REGION Network 2: ADD A STEP
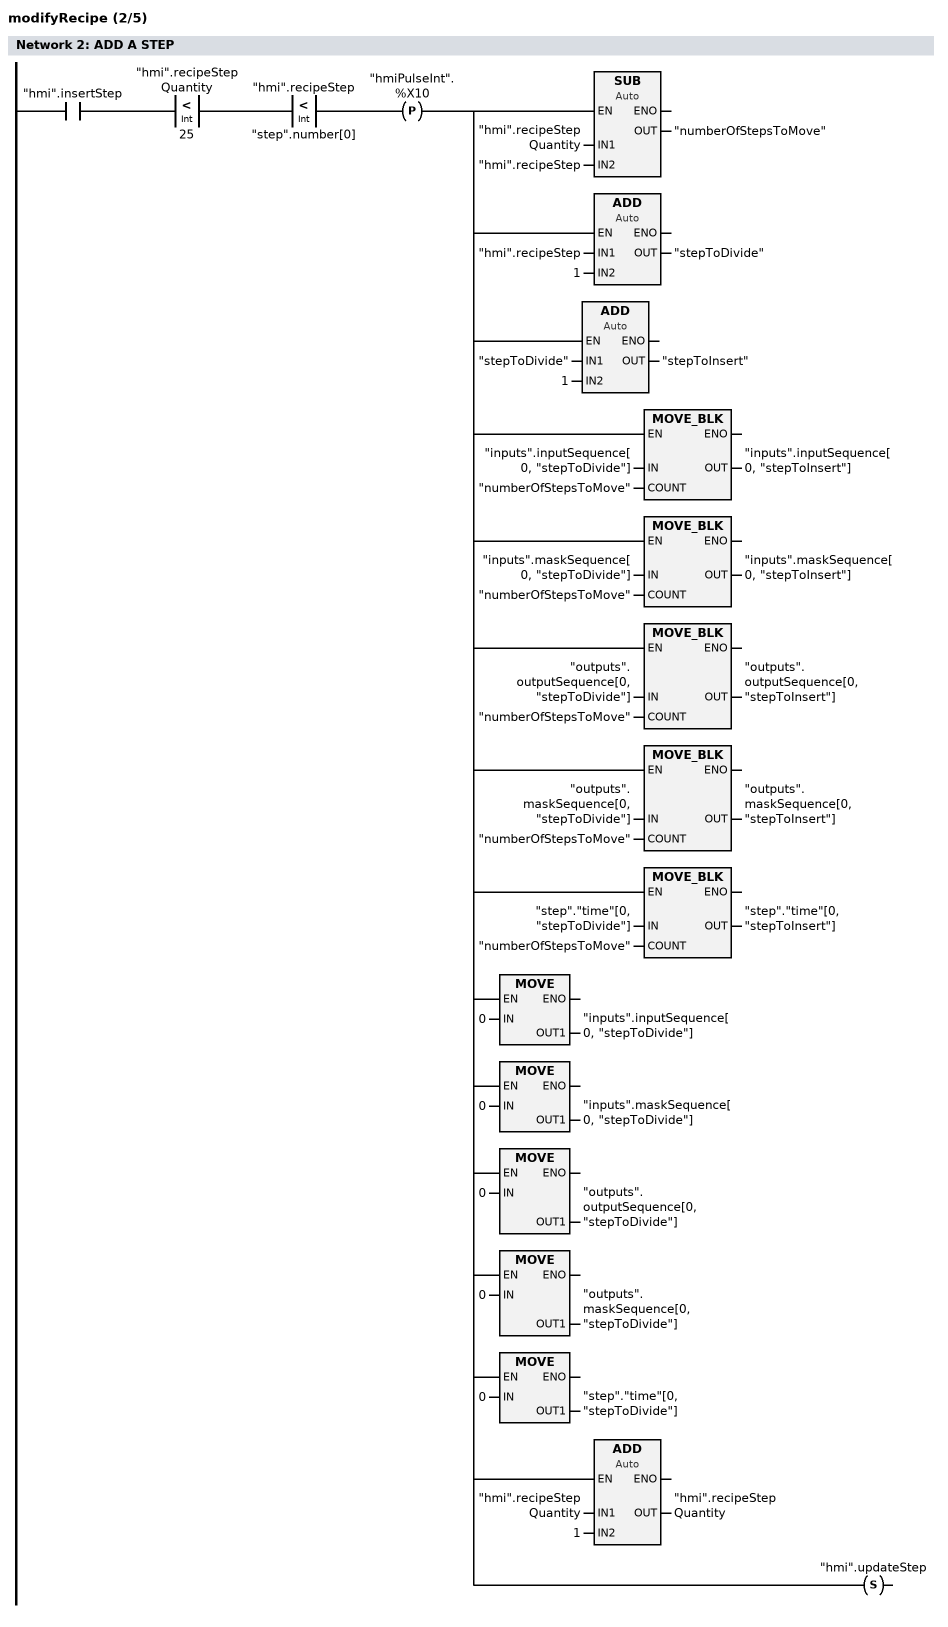
   #_w1 := "hmi".insertStep AND ("hmi".recipeStepQuantity < 25) AND ("hmi".recipeStep < "step".number[0]);
   #_w2 := #_w1 AND NOT "hmiPulseInt".%X10;   // rising edge
   "hmiPulseInt".%X10 := #_w1;
   IF #_w2 THEN
       "numberOfStepsToMove" := "hmi".recipeStepQuantity - "hmi".recipeStep;
       "stepToDivide" := "hmi".recipeStep + 1;
       "stepToInsert" := "stepToDivide" + 1;
       MOVE_BLK(IN := "inputs".inputSequence[0, "stepToDivide"],
                COUNT := "numberOfStepsToMove",
                OUT => "inputs".inputSequence[0, "stepToInsert"]);
       MOVE_BLK(IN := "inputs".maskSequence[0, "stepToDivide"],
                COUNT := "numberOfStepsToMove",
                OUT => "inputs".maskSequence[0, "stepToInsert"]);
       MOVE_BLK(IN := "outputs".outputSequence[0, "stepToDivide"],
                COUNT := "numberOfStepsToMove",
                OUT => "outputs".outputSequence[0, "stepToInsert"]);
       MOVE_BLK(IN := "outputs".maskSequence[0, "stepToDivide"],
                COUNT := "numberOfStepsToMove",
                OUT => "outputs".maskSequence[0, "stepToInsert"]);
       MOVE_BLK(IN := "step"."time"[0, "stepToDivide"],
                COUNT := "numberOfStepsToMove",
                OUT => "step"."time"[0, "stepToInsert"]);
       "inputs".inputSequence[0, "stepToDivide"] := 0;
       "inputs".maskSequence[0, "stepToDivide"] := 0;
       "outputs".outputSequence[0, "stepToDivide"] := 0;
       "outputs".maskSequence[0, "stepToDivide"] := 0;
       "step"."time"[0, "stepToDivide"] := 0;
       "hmi".recipeStepQuantity := "hmi".recipeStepQuantity + 1;
       "hmi".updateStep := TRUE;
   END_IF;
END_REGION

REGION Network 3: COPY A STEP
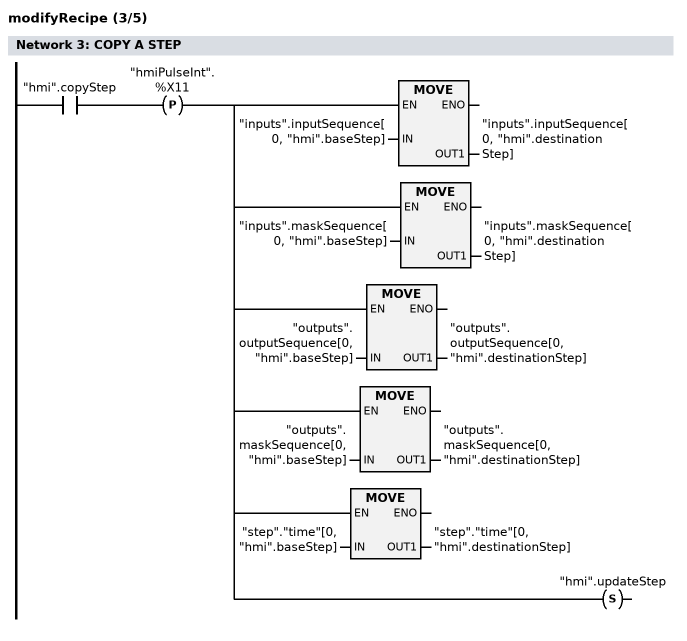
   RUNG wire#powerrail
      Contact( "hmi".copyStep )
      P_Trig( "hmiPulseInt".%X11 )
      wire#w1
      Move(in := "inputs".inputSequence[0, "hmi".baseStep], out1 => "inputs".inputSequence[0, "hmi".destinationStep])
   END_RUNG
   RUNG wire#w1
      Move(in := "inputs".maskSequence[0, "hmi".baseStep], out1 => "inputs".maskSequence[0, "hmi".destinationStep])
   END_RUNG
   RUNG wire#w1
      Move(in := "outputs".outputSequence[0, "hmi".baseStep], out1 => "outputs".outputSequence[0, "hmi".destinationStep])
   END_RUNG
   RUNG wire#w1
      Move(in := "outputs".maskSequence[0, "hmi".baseStep], out1 => "outputs".maskSequence[0, "hmi".destinationStep])
   END_RUNG
   RUNG wire#w1
      Move(in := "step"."time"[0, "hmi".baseStep], out1 => "step"."time"[0, "hmi".destinationStep])
   END_RUNG
   RUNG wire#w1
      S_Coil( "hmi".updateStep )
   END_RUNG
   // the same network as SCL:
   #_w1 := "hmi".copyStep AND NOT "hmiPulseInt".%X11;   // rising edge
   "hmiPulseInt".%X11 := "hmi".copyStep;
   IF #_w1 THEN
       "inputs".inputSequence[0, "hmi".destinationStep] := "inputs".inputSequence[0, "hmi".baseStep];
       "inputs".maskSequence[0, "hmi".destinationStep] := "inputs".maskSequence[0, "hmi".baseStep];
       "outputs".outputSequence[0, "hmi".destinationStep] := "outputs".outputSequence[0, "hmi".baseStep];
       "outputs".maskSequence[0, "hmi".destinationStep] := "outputs".maskSequence[0, "hmi".baseStep];
       "step"."time"[0, "hmi".destinationStep] := "step"."time"[0, "hmi".baseStep];
       "hmi".updateStep := TRUE;
   END_IF;
END_REGION

REGION Network 4: COPY SEQUENCE (COPY PART NUMBER)
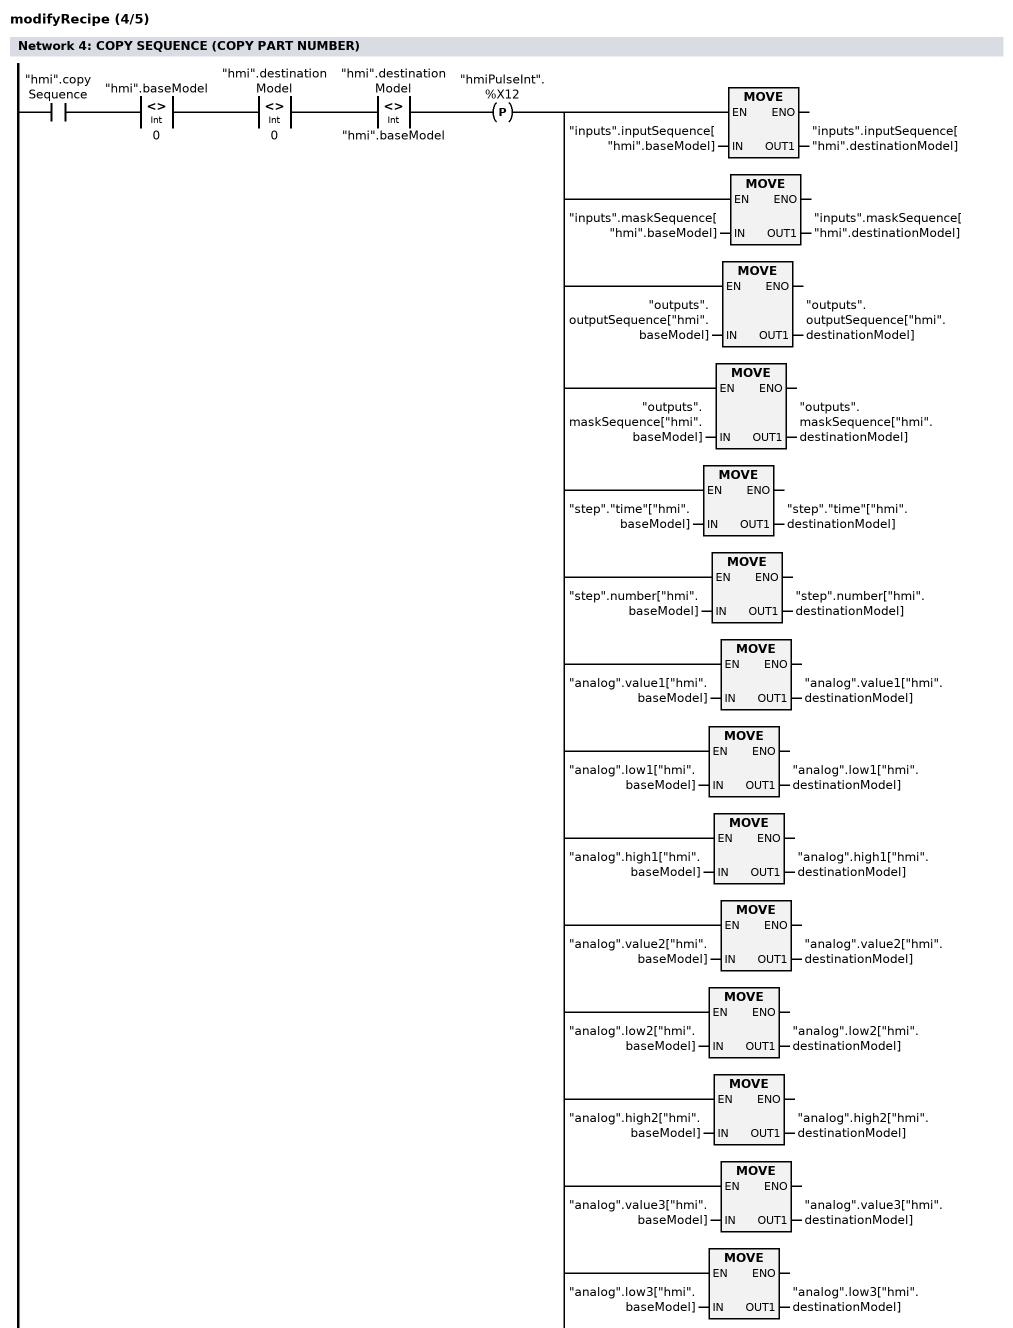
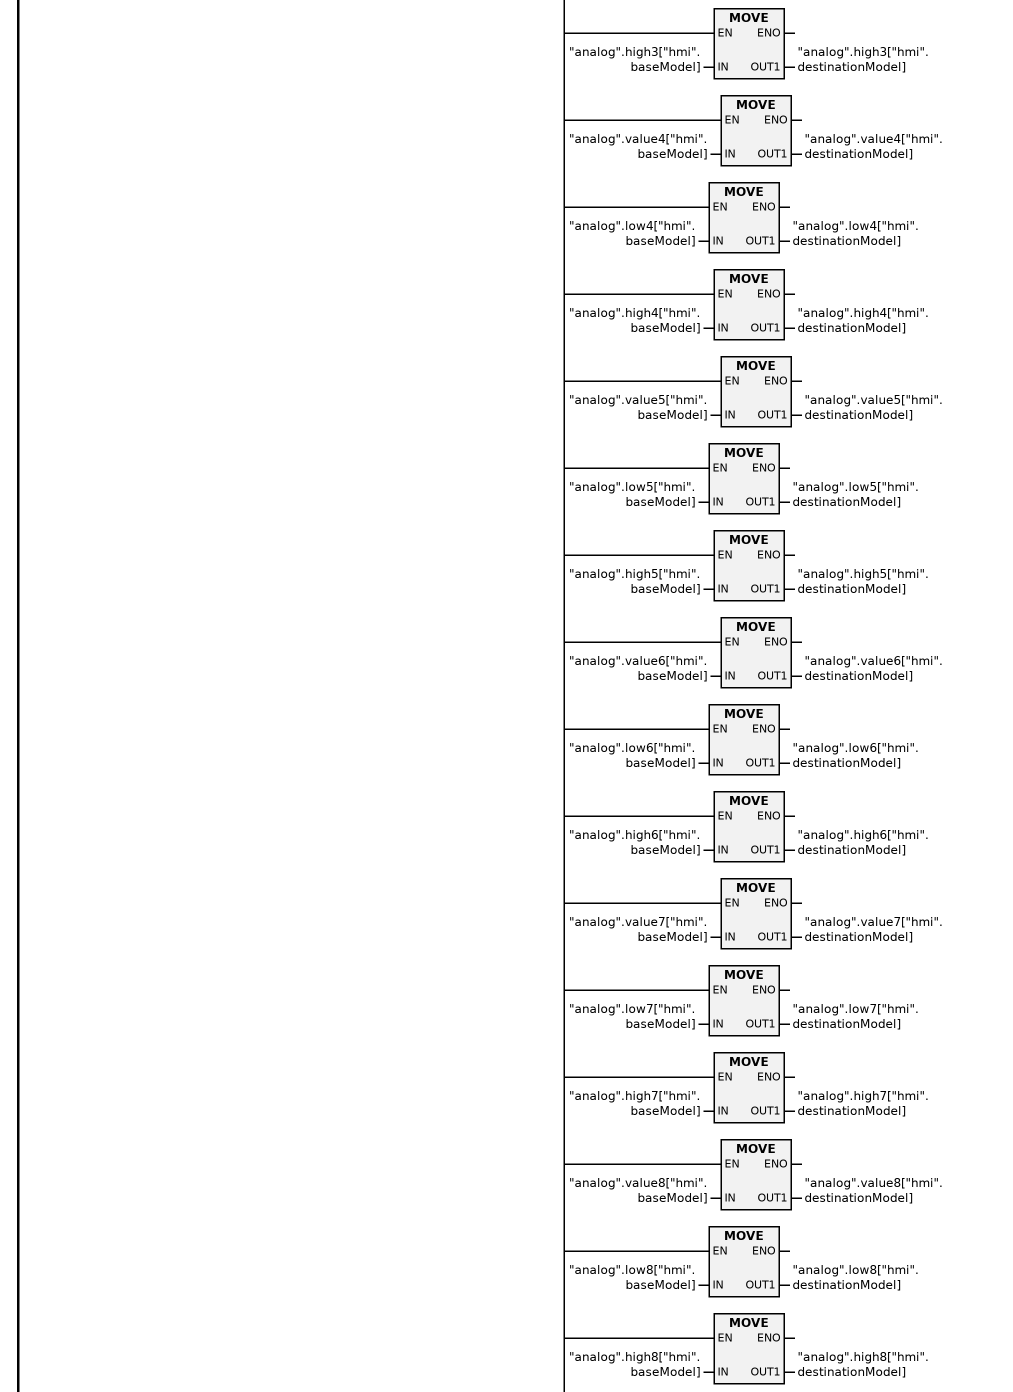
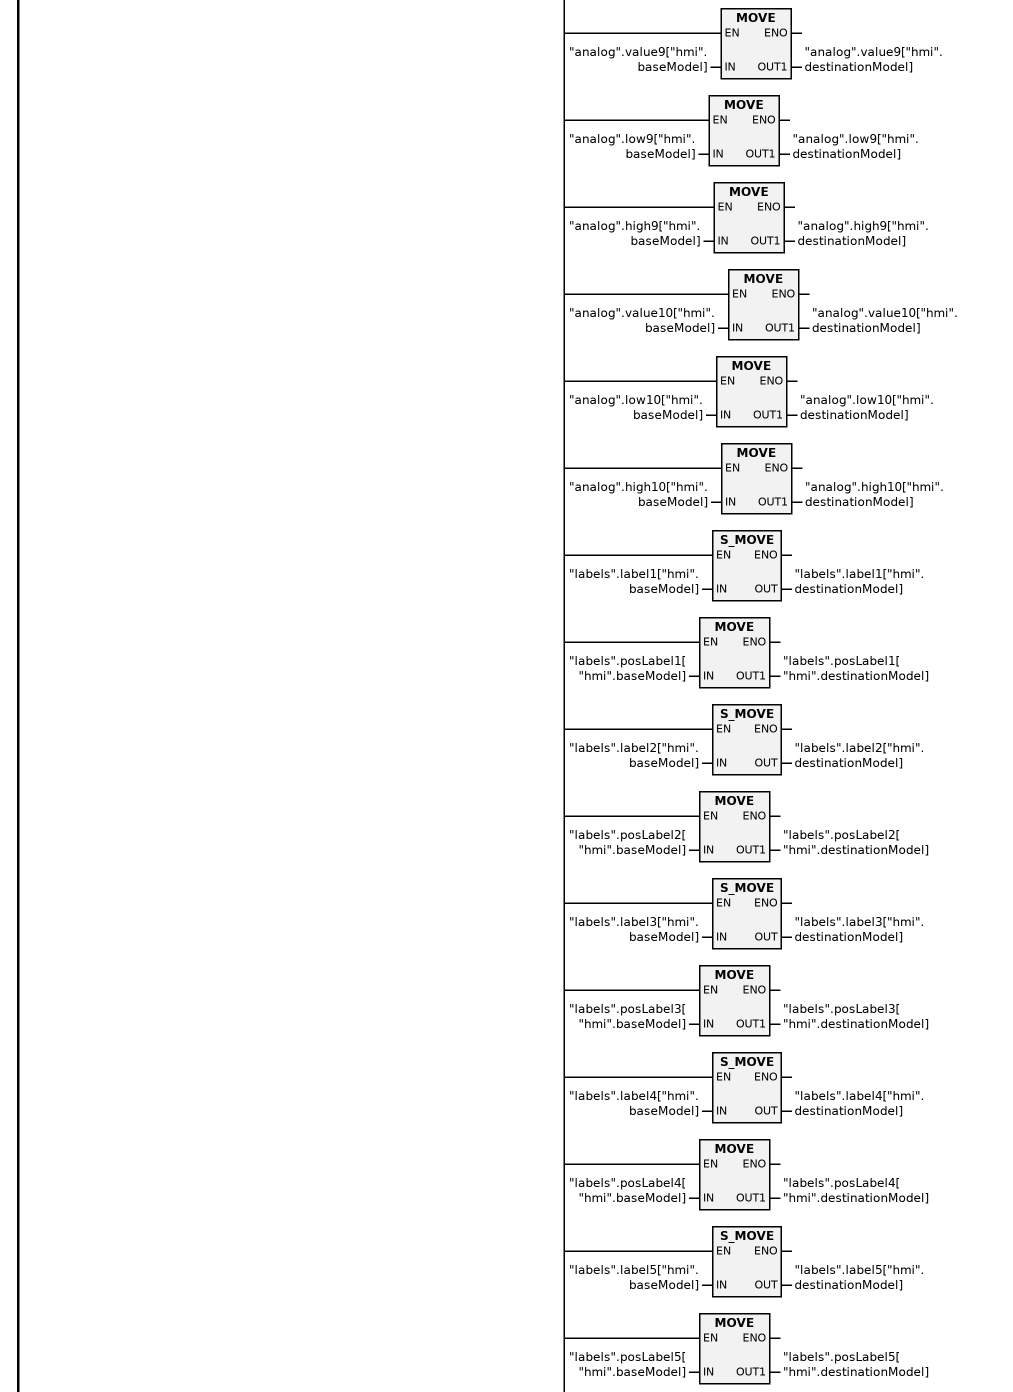
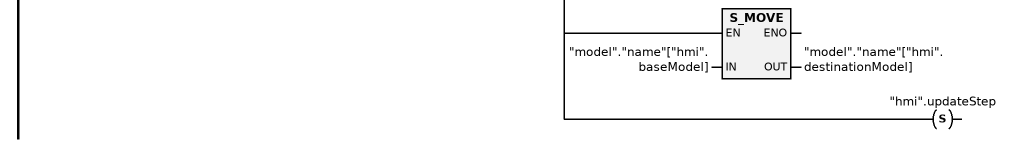
   RUNG wire#powerrail
      Contact( "hmi".copySequence )
      { S7_Templates := "SrcType := Int" } NE_Contact(in1 := "hmi".baseModel, in2 := 0)
      { S7_Templates := "SrcType := Int" } NE_Contact(in1 := "hmi".destinationModel, in2 := 0)
      { S7_Templates := "SrcType := Int" } NE_Contact(in1 := "hmi".destinationModel, in2 := "hmi".baseModel)
      P_Trig( "hmiPulseInt".%X12 )
      wire#w1
      Move(in := "inputs".inputSequence["hmi".baseModel], out1 => "inputs".inputSequence["hmi".destinationModel])
   END_RUNG
   RUNG wire#w1
      Move(in := "inputs".maskSequence["hmi".baseModel], out1 => "inputs".maskSequence["hmi".destinationModel])
   END_RUNG
   RUNG wire#w1
      Move(in := "outputs".outputSequence["hmi".baseModel], out1 => "outputs".outputSequence["hmi".destinationModel])
   END_RUNG
   RUNG wire#w1
      Move(in := "outputs".maskSequence["hmi".baseModel], out1 => "outputs".maskSequence["hmi".destinationModel])
   END_RUNG
   RUNG wire#w1
      Move(in := "step"."time"["hmi".baseModel], out1 => "step"."time"["hmi".destinationModel])
   END_RUNG
   RUNG wire#w1
      Move(in := "step".number["hmi".baseModel], out1 => "step".number["hmi".destinationModel])
   END_RUNG
   RUNG wire#w1
      Move(in := "analog".value1["hmi".baseModel], out1 => "analog".value1["hmi".destinationModel])
   END_RUNG
   RUNG wire#w1
      Move(in := "analog".low1["hmi".baseModel], out1 => "analog".low1["hmi".destinationModel])
   END_RUNG
   RUNG wire#w1
      Move(in := "analog".high1["hmi".baseModel], out1 => "analog".high1["hmi".destinationModel])
   END_RUNG
   RUNG wire#w1
      Move(in := "analog".value2["hmi".baseModel], out1 => "analog".value2["hmi".destinationModel])
   END_RUNG
   RUNG wire#w1
      Move(in := "analog".low2["hmi".baseModel], out1 => "analog".low2["hmi".destinationModel])
   END_RUNG
   RUNG wire#w1
      Move(in := "analog".high2["hmi".baseModel], out1 => "analog".high2["hmi".destinationModel])
   END_RUNG
   RUNG wire#w1
      Move(in := "analog".value3["hmi".baseModel], out1 => "analog".value3["hmi".destinationModel])
   END_RUNG
   RUNG wire#w1
      Move(in := "analog".low3["hmi".baseModel], out1 => "analog".low3["hmi".destinationModel])
   END_RUNG
   RUNG wire#w1
      Move(in := "analog".high3["hmi".baseModel], out1 => "analog".high3["hmi".destinationModel])
   END_RUNG
   RUNG wire#w1
      Move(in := "analog".value4["hmi".baseModel], out1 => "analog".value4["hmi".destinationModel])
   END_RUNG
   RUNG wire#w1
      Move(in := "analog".low4["hmi".baseModel], out1 => "analog".low4["hmi".destinationModel])
   END_RUNG
   RUNG wire#w1
      Move(in := "analog".high4["hmi".baseModel], out1 => "analog".high4["hmi".destinationModel])
   END_RUNG
   RUNG wire#w1
      Move(in := "analog".value5["hmi".baseModel], out1 => "analog".value5["hmi".destinationModel])
   END_RUNG
   RUNG wire#w1
      Move(in := "analog".low5["hmi".baseModel], out1 => "analog".low5["hmi".destinationModel])
   END_RUNG
   RUNG wire#w1
      Move(in := "analog".high5["hmi".baseModel], out1 => "analog".high5["hmi".destinationModel])
   END_RUNG
   RUNG wire#w1
      Move(in := "analog".value6["hmi".baseModel], out1 => "analog".value6["hmi".destinationModel])
   END_RUNG
   RUNG wire#w1
      Move(in := "analog".low6["hmi".baseModel], out1 => "analog".low6["hmi".destinationModel])
   END_RUNG
   RUNG wire#w1
      Move(in := "analog".high6["hmi".baseModel], out1 => "analog".high6["hmi".destinationModel])
   END_RUNG
   RUNG wire#w1
      Move(in := "analog".value7["hmi".baseModel], out1 => "analog".value7["hmi".destinationModel])
   END_RUNG
   RUNG wire#w1
      Move(in := "analog".low7["hmi".baseModel], out1 => "analog".low7["hmi".destinationModel])
   END_RUNG
   RUNG wire#w1
      Move(in := "analog".high7["hmi".baseModel], out1 => "analog".high7["hmi".destinationModel])
   END_RUNG
   RUNG wire#w1
      Move(in := "analog".value8["hmi".baseModel], out1 => "analog".value8["hmi".destinationModel])
   END_RUNG
   RUNG wire#w1
      Move(in := "analog".low8["hmi".baseModel], out1 => "analog".low8["hmi".destinationModel])
   END_RUNG
   RUNG wire#w1
      Move(in := "analog".high8["hmi".baseModel], out1 => "analog".high8["hmi".destinationModel])
   END_RUNG
   RUNG wire#w1
      Move(in := "analog".value9["hmi".baseModel], out1 => "analog".value9["hmi".destinationModel])
   END_RUNG
   RUNG wire#w1
      Move(in := "analog".low9["hmi".baseModel], out1 => "analog".low9["hmi".destinationModel])
   END_RUNG
   RUNG wire#w1
      Move(in := "analog".high9["hmi".baseModel], out1 => "analog".high9["hmi".destinationModel])
   END_RUNG
   RUNG wire#w1
      Move(in := "analog".value10["hmi".baseModel], out1 => "analog".value10["hmi".destinationModel])
   END_RUNG
   RUNG wire#w1
      Move(in := "analog".low10["hmi".baseModel], out1 => "analog".low10["hmi".destinationModel])
   END_RUNG
   RUNG wire#w1
      Move(in := "analog".high10["hmi".baseModel], out1 => "analog".high10["hmi".destinationModel])
   END_RUNG
   RUNG wire#w1
      S_Move(in := "labels".label1["hmi".baseModel], out => "labels".label1["hmi".destinationModel])
   END_RUNG
   RUNG wire#w1
      Move(in := "labels".posLabel1["hmi".baseModel], out1 => "labels".posLabel1["hmi".destinationModel])
   END_RUNG
   RUNG wire#w1
      S_Move(in := "labels".label2["hmi".baseModel], out => "labels".label2["hmi".destinationModel])
   END_RUNG
   RUNG wire#w1
      Move(in := "labels".posLabel2["hmi".baseModel], out1 => "labels".posLabel2["hmi".destinationModel])
   END_RUNG
   RUNG wire#w1
      S_Move(in := "labels".label3["hmi".baseModel], out => "labels".label3["hmi".destinationModel])
   END_RUNG
   RUNG wire#w1
      Move(in := "labels".posLabel3["hmi".baseModel], out1 => "labels".posLabel3["hmi".destinationModel])
   END_RUNG
   RUNG wire#w1
      S_Move(in := "labels".label4["hmi".baseModel], out => "labels".label4["hmi".destinationModel])
   END_RUNG
   RUNG wire#w1
      Move(in := "labels".posLabel4["hmi".baseModel], out1 => "labels".posLabel4["hmi".destinationModel])
   END_RUNG
   RUNG wire#w1
      S_Move(in := "labels".label5["hmi".baseModel], out => "labels".label5["hmi".destinationModel])
   END_RUNG
   RUNG wire#w1
      Move(in := "labels".posLabel5["hmi".baseModel], out1 => "labels".posLabel5["hmi".destinationModel])
   END_RUNG
   RUNG wire#w1
      S_Move(in := "model"."name"["hmi".baseModel], out => "model"."name"["hmi".destinationModel])
   END_RUNG
   RUNG wire#w1
      S_Coil( "hmi".updateStep )
   END_RUNG
   // the same network as SCL:
   #_w1 := "hmi".copySequence AND ("hmi".baseModel <> 0) AND ("hmi".destinationModel <> 0) AND ("hmi".destinationModel <> "hmi".baseModel);
   #_w2 := #_w1 AND NOT "hmiPulseInt".%X12;   // rising edge
   "hmiPulseInt".%X12 := #_w1;
   IF #_w2 THEN
       "inputs".inputSequence["hmi".destinationModel] := "inputs".inputSequence["hmi".baseModel];
       "inputs".maskSequence["hmi".destinationModel] := "inputs".maskSequence["hmi".baseModel];
       "outputs".outputSequence["hmi".destinationModel] := "outputs".outputSequence["hmi".baseModel];
       "outputs".maskSequence["hmi".destinationModel] := "outputs".maskSequence["hmi".baseModel];
       "step"."time"["hmi".destinationModel] := "step"."time"["hmi".baseModel];
       "step".number["hmi".destinationModel] := "step".number["hmi".baseModel];
       "analog".value1["hmi".destinationModel] := "analog".value1["hmi".baseModel];
       "analog".low1["hmi".destinationModel] := "analog".low1["hmi".baseModel];
       "analog".high1["hmi".destinationModel] := "analog".high1["hmi".baseModel];
       "analog".value2["hmi".destinationModel] := "analog".value2["hmi".baseModel];
       "analog".low2["hmi".destinationModel] := "analog".low2["hmi".baseModel];
       "analog".high2["hmi".destinationModel] := "analog".high2["hmi".baseModel];
       "analog".value3["hmi".destinationModel] := "analog".value3["hmi".baseModel];
       "analog".low3["hmi".destinationModel] := "analog".low3["hmi".baseModel];
       "analog".high3["hmi".destinationModel] := "analog".high3["hmi".baseModel];
       "analog".value4["hmi".destinationModel] := "analog".value4["hmi".baseModel];
       "analog".low4["hmi".destinationModel] := "analog".low4["hmi".baseModel];
       "analog".high4["hmi".destinationModel] := "analog".high4["hmi".baseModel];
       "analog".value5["hmi".destinationModel] := "analog".value5["hmi".baseModel];
       "analog".low5["hmi".destinationModel] := "analog".low5["hmi".baseModel];
       "analog".high5["hmi".destinationModel] := "analog".high5["hmi".baseModel];
       "analog".value6["hmi".destinationModel] := "analog".value6["hmi".baseModel];
       "analog".low6["hmi".destinationModel] := "analog".low6["hmi".baseModel];
       "analog".high6["hmi".destinationModel] := "analog".high6["hmi".baseModel];
       "analog".value7["hmi".destinationModel] := "analog".value7["hmi".baseModel];
       "analog".low7["hmi".destinationModel] := "analog".low7["hmi".baseModel];
       "analog".high7["hmi".destinationModel] := "analog".high7["hmi".baseModel];
       "analog".value8["hmi".destinationModel] := "analog".value8["hmi".baseModel];
       "analog".low8["hmi".destinationModel] := "analog".low8["hmi".baseModel];
       "analog".high8["hmi".destinationModel] := "analog".high8["hmi".baseModel];
       "analog".value9["hmi".destinationModel] := "analog".value9["hmi".baseModel];
       "analog".low9["hmi".destinationModel] := "analog".low9["hmi".baseModel];
       "analog".high9["hmi".destinationModel] := "analog".high9["hmi".baseModel];
       "analog".value10["hmi".destinationModel] := "analog".value10["hmi".baseModel];
       "analog".low10["hmi".destinationModel] := "analog".low10["hmi".baseModel];
       "analog".high10["hmi".destinationModel] := "analog".high10["hmi".baseModel];
       "labels".label1["hmi".destinationModel] := "labels".label1["hmi".baseModel];
       "labels".posLabel1["hmi".destinationModel] := "labels".posLabel1["hmi".baseModel];
       "labels".label2["hmi".destinationModel] := "labels".label2["hmi".baseModel];
       "labels".posLabel2["hmi".destinationModel] := "labels".posLabel2["hmi".baseModel];
       "labels".label3["hmi".destinationModel] := "labels".label3["hmi".baseModel];
       "labels".posLabel3["hmi".destinationModel] := "labels".posLabel3["hmi".baseModel];
       "labels".label4["hmi".destinationModel] := "labels".label4["hmi".baseModel];
       "labels".posLabel4["hmi".destinationModel] := "labels".posLabel4["hmi".baseModel];
       "labels".label5["hmi".destinationModel] := "labels".label5["hmi".baseModel];
       "labels".posLabel5["hmi".destinationModel] := "labels".posLabel5["hmi".baseModel];
       "model"."name"["hmi".destinationModel] := "model"."name"["hmi".baseModel];
       "hmi".updateStep := TRUE;
   END_IF;
END_REGION

REGION Network 5: COPY A STEP (#) FROM A PROGRAM (#) IN ANOTHER STEP (#) FROM ANOTHER PROGRAM (#)
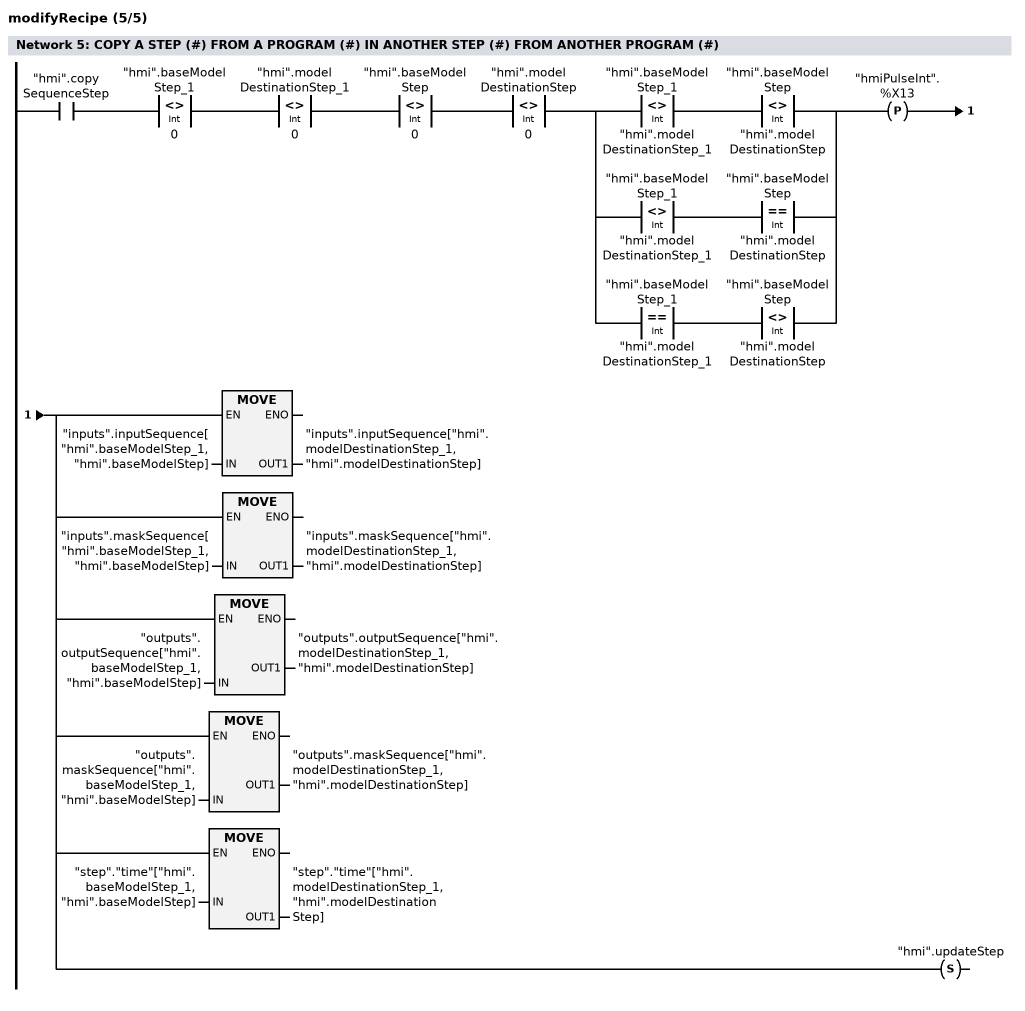
   RUNG wire#powerrail
      Contact( "hmi".copySequenceStep )
      { S7_Templates := "SrcType := Int" } NE_Contact(in1 := "hmi".baseModelStep_1, in2 := 0)
      { S7_Templates := "SrcType := Int" } NE_Contact(in1 := "hmi".modelDestinationStep_1, in2 := 0)
      { S7_Templates := "SrcType := Int" } NE_Contact(in1 := "hmi".baseModelStep, in2 := 0)
      { S7_Templates := "SrcType := Int" } NE_Contact(in1 := "hmi".modelDestinationStep, in2 := 0)
      wire#w1
      { S7_Templates := "SrcType := Int" } NE_Contact(in1 := "hmi".baseModelStep_1, in2 := "hmi".modelDestinationStep_1)
      { S7_Templates := "SrcType := Int" } NE_Contact(in1 := "hmi".baseModelStep, in2 := "hmi".modelDestinationStep)
      wire#w2
      P_Trig( "hmiPulseInt".%X13 )
      wire#w3
      Move(in := "inputs".inputSequence["hmi".baseModelStep_1, "hmi".baseModelStep], out1 => "inputs".inputSequence["hmi".modelDestinationStep_1, "hmi".modelDestinationStep])
   END_RUNG
   RUNG wire#w1
      { S7_Templates := "SrcType := Int" } NE_Contact(in1 := "hmi".baseModelStep_1, in2 := "hmi".modelDestinationStep_1)
      { S7_Templates := "SrcType := Int" } EQ_Contact(in1 := "hmi".baseModelStep, in2 := "hmi".modelDestinationStep)
   END_RUNG wire#w2
   RUNG wire#w1
      { S7_Templates := "SrcType := Int" } EQ_Contact(in1 := "hmi".baseModelStep_1, in2 := "hmi".modelDestinationStep_1)
      { S7_Templates := "SrcType := Int" } NE_Contact(in1 := "hmi".baseModelStep, in2 := "hmi".modelDestinationStep)
   END_RUNG wire#w2
   RUNG wire#w3
      Move(in := "inputs".maskSequence["hmi".baseModelStep_1, "hmi".baseModelStep], out1 => "inputs".maskSequence["hmi".modelDestinationStep_1, "hmi".modelDestinationStep])
   END_RUNG
   RUNG wire#w3
      Move(in := "outputs".outputSequence["hmi".baseModelStep_1, "hmi".baseModelStep], out1 => "outputs".outputSequence["hmi".modelDestinationStep_1, "hmi".modelDestinationStep])
   END_RUNG
   RUNG wire#w3
      Move(in := "outputs".maskSequence["hmi".baseModelStep_1, "hmi".baseModelStep], out1 => "outputs".maskSequence["hmi".modelDestinationStep_1, "hmi".modelDestinationStep])
   END_RUNG
   RUNG wire#w3
      Move(in := "step"."time"["hmi".baseModelStep_1, "hmi".baseModelStep], out1 => "step"."time"["hmi".modelDestinationStep_1, "hmi".modelDestinationStep])
   END_RUNG
   RUNG wire#w3
      S_Coil( "hmi".updateStep )
   END_RUNG
   // the same network as SCL:
   #_w1 := "hmi".copySequenceStep AND ("hmi".baseModelStep_1 <> 0) AND ("hmi".modelDestinationStep_1 <> 0) AND ("hmi".baseModelStep <> 0) AND ("hmi".modelDestinationStep <> 0) AND ((("hmi".baseModelStep_1 <> "hmi".modelDestinationStep_1) AND ("hmi".baseModelStep <> "hmi".modelDestinationStep)) OR (("hmi".baseModelStep_1 <> "hmi".modelDestinationStep_1) AND ("hmi".baseModelStep = "hmi".modelDestinationStep)) OR (("hmi".baseModelStep_1 = "hmi".modelDestinationStep_1) AND ("hmi".baseModelStep <> "hmi".modelDestinationStep)));
   #_w2 := #_w1 AND NOT "hmiPulseInt".%X13;   // rising edge
   "hmiPulseInt".%X13 := #_w1;
   IF #_w2 THEN
       "inputs".inputSequence["hmi".modelDestinationStep_1, "hmi".modelDestinationStep] := "inputs".inputSequence["hmi".baseModelStep_1, "hmi".baseModelStep];
       "inputs".maskSequence["hmi".modelDestinationStep_1, "hmi".modelDestinationStep] := "inputs".maskSequence["hmi".baseModelStep_1, "hmi".baseModelStep];
       "outputs".outputSequence["hmi".modelDestinationStep_1, "hmi".modelDestinationStep] := "outputs".outputSequence["hmi".baseModelStep_1, "hmi".baseModelStep];
       "outputs".maskSequence["hmi".modelDestinationStep_1, "hmi".modelDestinationStep] := "outputs".maskSequence["hmi".baseModelStep_1, "hmi".baseModelStep];
       "step"."time"["hmi".modelDestinationStep_1, "hmi".modelDestinationStep] := "step"."time"["hmi".baseModelStep_1, "hmi".baseModelStep];
       "hmi".updateStep := TRUE;
   END_IF;
END_REGION
END_FUNCTION

FUNCTION "inputsMapping" : Void   // FC1, LAD
{ S7_Optimized_Access := 'TRUE' }
VERSION : 0.1
// stored: AutoNumber true, IsIECCheckEnabled false, SetENOAutomatically false, UDAEnableTagReadback false
BEGIN

REGION Network 1: A00.- Clear Data
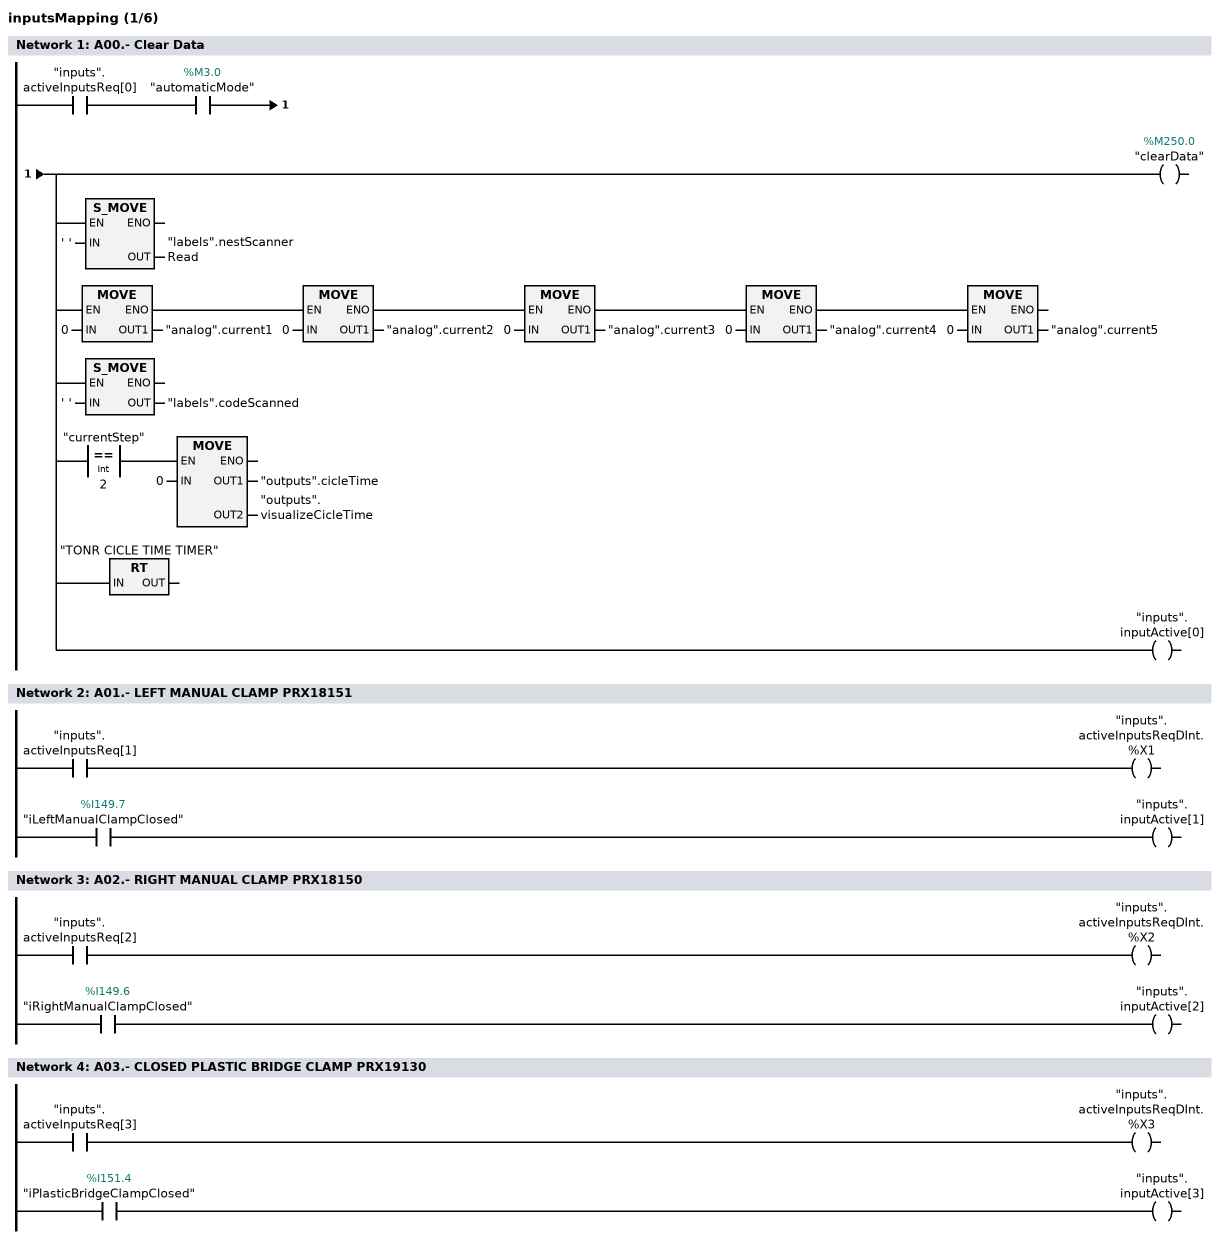
   RUNG wire#powerrail
      Contact( "inputs".activeInputsReq[0] )
      Contact( "automaticMode" )
      wire#w1
      Coil( "clearData" )
   END_RUNG
   RUNG wire#w1
      S_Move(in := ' ', out => "labels".nestScannerRead)
   END_RUNG
   RUNG wire#w1
      Move(in := 0, out1 => "analog".current1)
      Move(in := 0, out1 => "analog".current2)
      Move(in := 0, out1 => "analog".current3)
      Move(in := 0, out1 => "analog".current4)
      Move(in := 0, out1 => "analog".current5)
   END_RUNG
   RUNG wire#w1
      S_Move(in := ' ', out => "labels".codeScanned)
   END_RUNG
   RUNG wire#w1
      { S7_Templates := "SrcType := Int" } EQ_Contact(in1 := "currentStep", in2 := 2)
      Move(in := 0, out1 => "outputs".cicleTime, out2 => "outputs".visualizeCicleTime)
   END_RUNG
   RUNG wire#w1
      RT_Coil( "TONR CICLE TIME TIMER" )
   END_RUNG
   RUNG wire#w1
      Coil( "inputs".inputActive[0] )
   END_RUNG
   // the same network as SCL:
   "clearData" := "inputs".activeInputsReq[0] AND "automaticMode";
   IF "clearData" THEN
       "labels".nestScannerRead := ' ';
       "analog".current1 := 0;
       "analog".current2 := 0;
       "analog".current3 := 0;
       "analog".current4 := 0;
       "analog".current5 := 0;
       "labels".codeScanned := ' ';
   END_IF;
   IF "clearData" AND ("currentStep" = 2) THEN
       "outputs".cicleTime := 0;
       "outputs".visualizeCicleTime := 0;
   END_IF;
   IF "clearData" THEN RESET_TIMER("TONR CICLE TIME TIMER"); END_IF;
   "inputs".inputActive[0] := "clearData";
END_REGION

REGION Network 2: A01.- LEFT MANUAL CLAMP PRX18151
   RUNG wire#powerrail
      Contact( "inputs".activeInputsReq[1] )
      Coil( "inputs".activeInputsReqDInt.%X1 )
   END_RUNG
   RUNG wire#powerrail
      Contact( "iLeftManualClampClosed" )
      Coil( "inputs".inputActive[1] )
   END_RUNG
   // the same network as SCL:
   "inputs".activeInputsReqDInt.%X1 := "inputs".activeInputsReq[1];
   "inputs".inputActive[1] := "iLeftManualClampClosed";
END_REGION

REGION Network 3: A02.- RIGHT MANUAL CLAMP PRX18150
   RUNG wire#powerrail
      Contact( "inputs".activeInputsReq[2] )
      Coil( "inputs".activeInputsReqDInt.%X2 )
   END_RUNG
   RUNG wire#powerrail
      Contact( "iRightManualClampClosed" )
      Coil( "inputs".inputActive[2] )
   END_RUNG
   // the same network as SCL:
   "inputs".activeInputsReqDInt.%X2 := "inputs".activeInputsReq[2];
   "inputs".inputActive[2] := "iRightManualClampClosed";
END_REGION

REGION Network 4: A03.- CLOSED PLASTIC BRIDGE CLAMP PRX19130
   RUNG wire#powerrail
      Contact( "inputs".activeInputsReq[3] )
      Coil( "inputs".activeInputsReqDInt.%X3 )
   END_RUNG
   RUNG wire#powerrail
      Contact( "iPlasticBridgeClampClosed" )
      Coil( "inputs".inputActive[3] )
   END_RUNG
   // the same network as SCL:
   "inputs".activeInputsReqDInt.%X3 := "inputs".activeInputsReq[3];
   "inputs".inputActive[3] := "iPlasticBridgeClampClosed";
END_REGION

REGION Network 5: A04.- PLASTIC BRIDGE PRESENT PRX19090
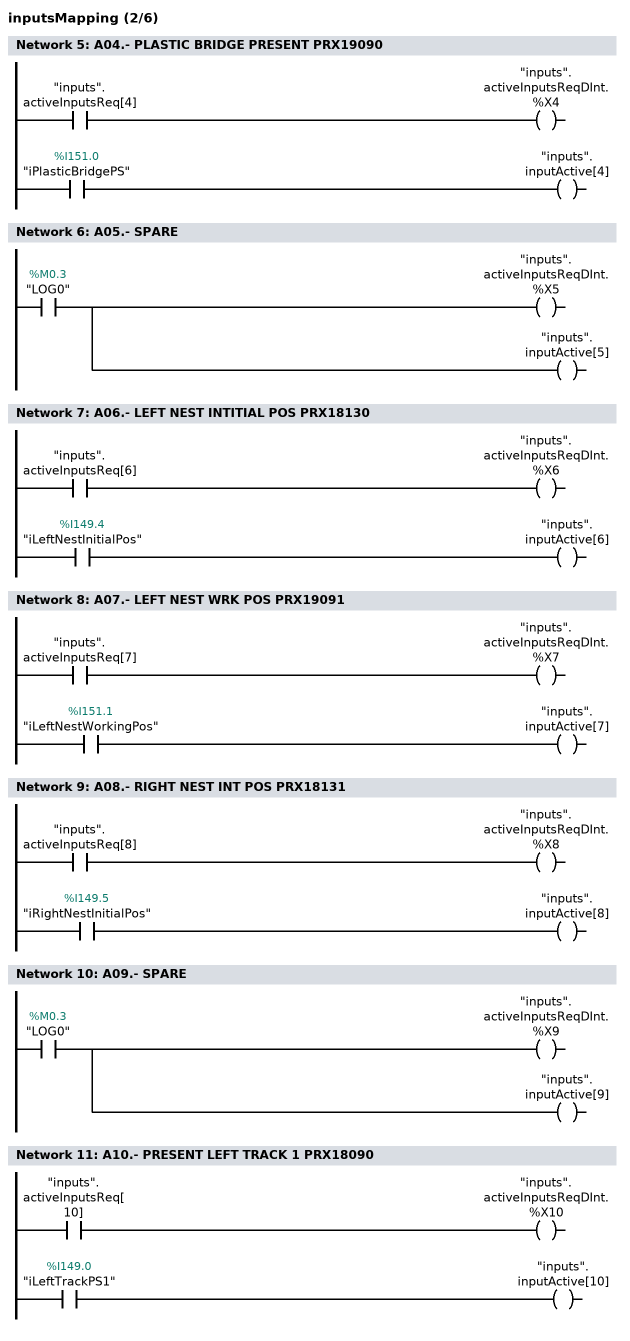
   RUNG wire#powerrail
      Contact( "inputs".activeInputsReq[4] )
      Coil( "inputs".activeInputsReqDInt.%X4 )
   END_RUNG
   RUNG wire#powerrail
      Contact( "iPlasticBridgePS" )
      Coil( "inputs".inputActive[4] )
   END_RUNG
   // the same network as SCL:
   "inputs".activeInputsReqDInt.%X4 := "inputs".activeInputsReq[4];
   "inputs".inputActive[4] := "iPlasticBridgePS";
END_REGION

REGION Network 6: A05.- SPARE
   RUNG wire#powerrail
      Contact( "LOG0" )
      wire#w1
      Coil( "inputs".activeInputsReqDInt.%X5 )
   END_RUNG
   RUNG wire#w1
      Coil( "inputs".inputActive[5] )
   END_RUNG
   // the same network as SCL:
   "inputs".activeInputsReqDInt.%X5 := "LOG0";
   "inputs".inputActive[5] := "LOG0";
END_REGION

REGION Network 7: A06.- LEFT NEST INTITIAL POS PRX18130
   RUNG wire#powerrail
      Contact( "inputs".activeInputsReq[6] )
      Coil( "inputs".activeInputsReqDInt.%X6 )
   END_RUNG
   RUNG wire#powerrail
      Contact( "iLeftNestInitialPos" )
      Coil( "inputs".inputActive[6] )
   END_RUNG
   // the same network as SCL:
   "inputs".activeInputsReqDInt.%X6 := "inputs".activeInputsReq[6];
   "inputs".inputActive[6] := "iLeftNestInitialPos";
END_REGION

REGION Network 8: A07.- LEFT NEST WRK POS PRX19091
   RUNG wire#powerrail
      Contact( "inputs".activeInputsReq[7] )
      Coil( "inputs".activeInputsReqDInt.%X7 )
   END_RUNG
   RUNG wire#powerrail
      Contact( "iLeftNestWorkingPos" )
      Coil( "inputs".inputActive[7] )
   END_RUNG
   // the same network as SCL:
   "inputs".activeInputsReqDInt.%X7 := "inputs".activeInputsReq[7];
   "inputs".inputActive[7] := "iLeftNestWorkingPos";
END_REGION

REGION Network 9: A08.- RIGHT NEST INT POS PRX18131
   RUNG wire#powerrail
      Contact( "inputs".activeInputsReq[8] )
      Coil( "inputs".activeInputsReqDInt.%X8 )
   END_RUNG
   RUNG wire#powerrail
      Contact( "iRightNestInitialPos" )
      Coil( "inputs".inputActive[8] )
   END_RUNG
   // the same network as SCL:
   "inputs".activeInputsReqDInt.%X8 := "inputs".activeInputsReq[8];
   "inputs".inputActive[8] := "iRightNestInitialPos";
END_REGION

REGION Network 10: A09.- SPARE
   RUNG wire#powerrail
      Contact( "LOG0" )
      wire#w1
      Coil( "inputs".activeInputsReqDInt.%X9 )
   END_RUNG
   RUNG wire#w1
      Coil( "inputs".inputActive[9] )
   END_RUNG
   // the same network as SCL:
   "inputs".activeInputsReqDInt.%X9 := "LOG0";
   "inputs".inputActive[9] := "LOG0";
END_REGION

REGION Network 11: A10.- PRESENT LEFT TRACK 1 PRX18090
   RUNG wire#powerrail
      Contact( "inputs".activeInputsReq[10] )
      Coil( "inputs".activeInputsReqDInt.%X10 )
   END_RUNG
   RUNG wire#powerrail
      Contact( "iLeftTrackPS1" )
      Coil( "inputs".inputActive[10] )
   END_RUNG
   // the same network as SCL:
   "inputs".activeInputsReqDInt.%X10 := "inputs".activeInputsReq[10];
   "inputs".inputActive[10] := "iLeftTrackPS1";
END_REGION

REGION Network 12: A11.- PRESENT RIGHT TRACK 1 PRX18110
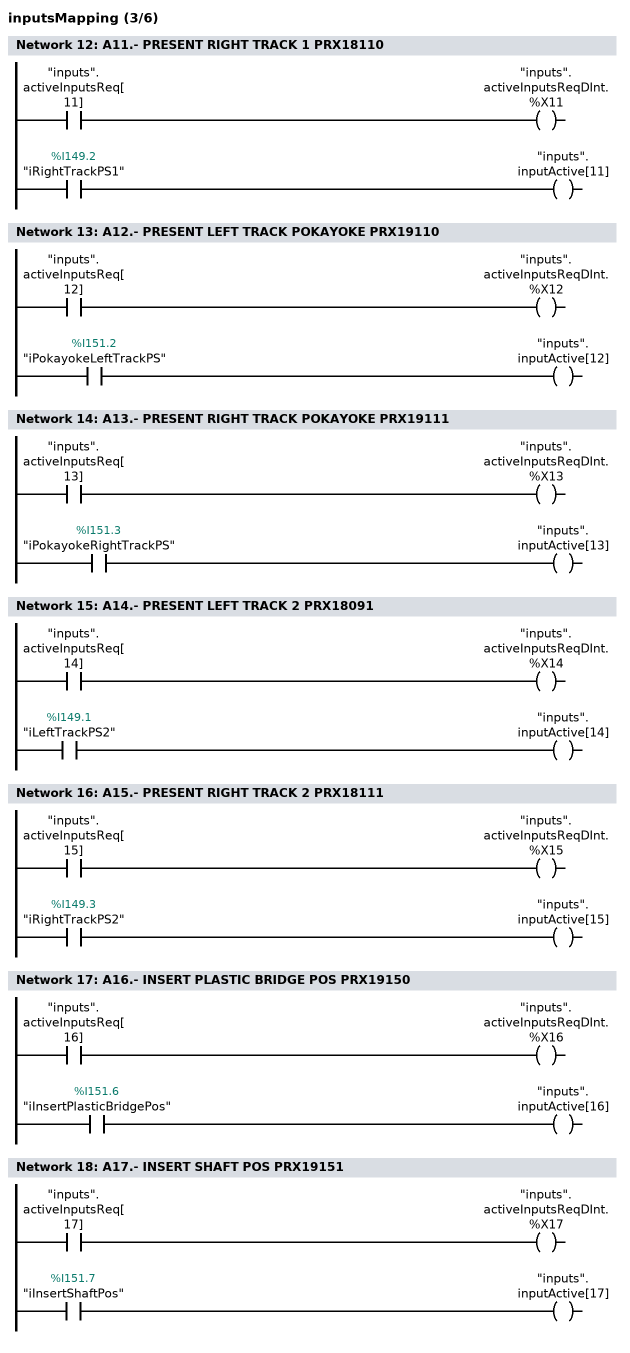
   RUNG wire#powerrail
      Contact( "inputs".activeInputsReq[11] )
      Coil( "inputs".activeInputsReqDInt.%X11 )
   END_RUNG
   RUNG wire#powerrail
      Contact( "iRightTrackPS1" )
      Coil( "inputs".inputActive[11] )
   END_RUNG
   // the same network as SCL:
   "inputs".activeInputsReqDInt.%X11 := "inputs".activeInputsReq[11];
   "inputs".inputActive[11] := "iRightTrackPS1";
END_REGION

REGION Network 13: A12.- PRESENT LEFT TRACK POKAYOKE PRX19110
   RUNG wire#powerrail
      Contact( "inputs".activeInputsReq[12] )
      Coil( "inputs".activeInputsReqDInt.%X12 )
   END_RUNG
   RUNG wire#powerrail
      Contact( "iPokayokeLeftTrackPS" )
      Coil( "inputs".inputActive[12] )
   END_RUNG
   // the same network as SCL:
   "inputs".activeInputsReqDInt.%X12 := "inputs".activeInputsReq[12];
   "inputs".inputActive[12] := "iPokayokeLeftTrackPS";
END_REGION

REGION Network 14: A13.- PRESENT RIGHT TRACK POKAYOKE PRX19111
   RUNG wire#powerrail
      Contact( "inputs".activeInputsReq[13] )
      Coil( "inputs".activeInputsReqDInt.%X13 )
   END_RUNG
   RUNG wire#powerrail
      Contact( "iPokayokeRightTrackPS" )
      Coil( "inputs".inputActive[13] )
   END_RUNG
   // the same network as SCL:
   "inputs".activeInputsReqDInt.%X13 := "inputs".activeInputsReq[13];
   "inputs".inputActive[13] := "iPokayokeRightTrackPS";
END_REGION

REGION Network 15: A14.- PRESENT LEFT TRACK 2 PRX18091
   RUNG wire#powerrail
      Contact( "inputs".activeInputsReq[14] )
      Coil( "inputs".activeInputsReqDInt.%X14 )
   END_RUNG
   RUNG wire#powerrail
      Contact( "iLeftTrackPS2" )
      Coil( "inputs".inputActive[14] )
   END_RUNG
   // the same network as SCL:
   "inputs".activeInputsReqDInt.%X14 := "inputs".activeInputsReq[14];
   "inputs".inputActive[14] := "iLeftTrackPS2";
END_REGION

REGION Network 16: A15.- PRESENT RIGHT TRACK 2 PRX18111
   RUNG wire#powerrail
      Contact( "inputs".activeInputsReq[15] )
      Coil( "inputs".activeInputsReqDInt.%X15 )
   END_RUNG
   RUNG wire#powerrail
      Contact( "iRightTrackPS2" )
      Coil( "inputs".inputActive[15] )
   END_RUNG
   // the same network as SCL:
   "inputs".activeInputsReqDInt.%X15 := "inputs".activeInputsReq[15];
   "inputs".inputActive[15] := "iRightTrackPS2";
END_REGION

REGION Network 17: A16.- INSERT PLASTIC BRIDGE POS PRX19150
   RUNG wire#powerrail
      Contact( "inputs".activeInputsReq[16] )
      Coil( "inputs".activeInputsReqDInt.%X16 )
   END_RUNG
   RUNG wire#powerrail
      Contact( "iInsertPlasticBridgePos" )
      Coil( "inputs".inputActive[16] )
   END_RUNG
   // the same network as SCL:
   "inputs".activeInputsReqDInt.%X16 := "inputs".activeInputsReq[16];
   "inputs".inputActive[16] := "iInsertPlasticBridgePos";
END_REGION

REGION Network 18: A17.- INSERT SHAFT POS PRX19151
   RUNG wire#powerrail
      Contact( "inputs".activeInputsReq[17] )
      Coil( "inputs".activeInputsReqDInt.%X17 )
   END_RUNG
   RUNG wire#powerrail
      Contact( "iInsertShaftPos" )
      Coil( "inputs".inputActive[17] )
   END_RUNG
   // the same network as SCL:
   "inputs".activeInputsReqDInt.%X17 := "inputs".activeInputsReq[17];
   "inputs".inputActive[17] := "iInsertShaftPos";
END_REGION

REGION Network 19: A18.- REMOVE PIECE
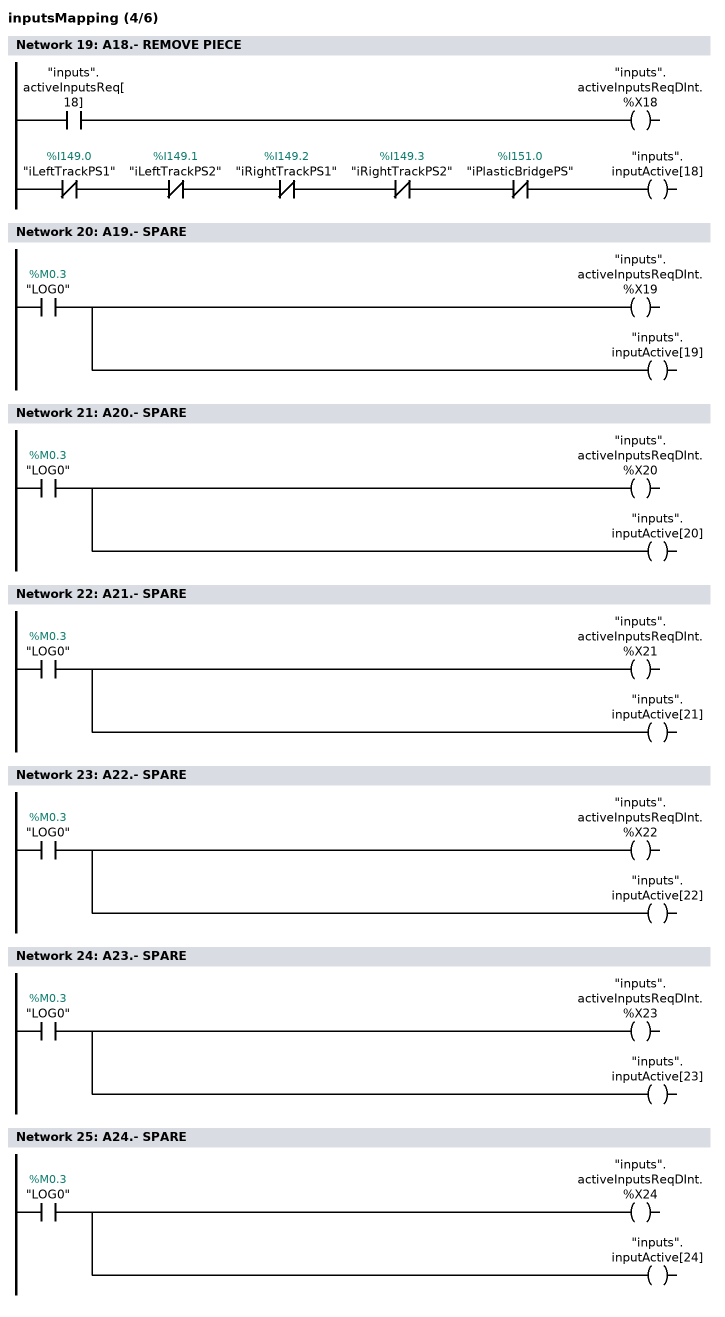
   RUNG wire#powerrail
      Contact( "inputs".activeInputsReq[18] )
      Coil( "inputs".activeInputsReqDInt.%X18 )
   END_RUNG
   RUNG wire#powerrail
      I_Contact( "iLeftTrackPS1" )
      I_Contact( "iLeftTrackPS2" )
      I_Contact( "iRightTrackPS1" )
      I_Contact( "iRightTrackPS2" )
      I_Contact( "iPlasticBridgePS" )
      Coil( "inputs".inputActive[18] )
   END_RUNG
   // the same network as SCL:
   "inputs".activeInputsReqDInt.%X18 := "inputs".activeInputsReq[18];
   "inputs".inputActive[18] := NOT "iLeftTrackPS1" AND NOT "iLeftTrackPS2" AND NOT "iRightTrackPS1" AND NOT "iRightTrackPS2" AND NOT "iPlasticBridgePS";
END_REGION

REGION Network 20: A19.- SPARE
   RUNG wire#powerrail
      Contact( "LOG0" )
      wire#w1
      Coil( "inputs".activeInputsReqDInt.%X19 )
   END_RUNG
   RUNG wire#w1
      Coil( "inputs".inputActive[19] )
   END_RUNG
   // the same network as SCL:
   "inputs".activeInputsReqDInt.%X19 := "LOG0";
   "inputs".inputActive[19] := "LOG0";
END_REGION

REGION Network 21: A20.- SPARE
   RUNG wire#powerrail
      Contact( "LOG0" )
      wire#w1
      Coil( "inputs".activeInputsReqDInt.%X20 )
   END_RUNG
   RUNG wire#w1
      Coil( "inputs".inputActive[20] )
   END_RUNG
   // the same network as SCL:
   "inputs".activeInputsReqDInt.%X20 := "LOG0";
   "inputs".inputActive[20] := "LOG0";
END_REGION

REGION Network 22: A21.- SPARE
   RUNG wire#powerrail
      Contact( "LOG0" )
      wire#w1
      Coil( "inputs".activeInputsReqDInt.%X21 )
   END_RUNG
   RUNG wire#w1
      Coil( "inputs".inputActive[21] )
   END_RUNG
   // the same network as SCL:
   "inputs".activeInputsReqDInt.%X21 := "LOG0";
   "inputs".inputActive[21] := "LOG0";
END_REGION

REGION Network 23: A22.- SPARE
   RUNG wire#powerrail
      Contact( "LOG0" )
      wire#w1
      Coil( "inputs".activeInputsReqDInt.%X22 )
   END_RUNG
   RUNG wire#w1
      Coil( "inputs".inputActive[22] )
   END_RUNG
   // the same network as SCL:
   "inputs".activeInputsReqDInt.%X22 := "LOG0";
   "inputs".inputActive[22] := "LOG0";
END_REGION

REGION Network 24: A23.- SPARE
   RUNG wire#powerrail
      Contact( "LOG0" )
      wire#w1
      Coil( "inputs".activeInputsReqDInt.%X23 )
   END_RUNG
   RUNG wire#w1
      Coil( "inputs".inputActive[23] )
   END_RUNG
   // the same network as SCL:
   "inputs".activeInputsReqDInt.%X23 := "LOG0";
   "inputs".inputActive[23] := "LOG0";
END_REGION

REGION Network 25: A24.- SPARE
   RUNG wire#powerrail
      Contact( "LOG0" )
      wire#w1
      Coil( "inputs".activeInputsReqDInt.%X24 )
   END_RUNG
   RUNG wire#w1
      Coil( "inputs".inputActive[24] )
   END_RUNG
   // the same network as SCL:
   "inputs".activeInputsReqDInt.%X24 := "LOG0";
   "inputs".inputActive[24] := "LOG0";
END_REGION

REGION Network 26: A25.- SPARE
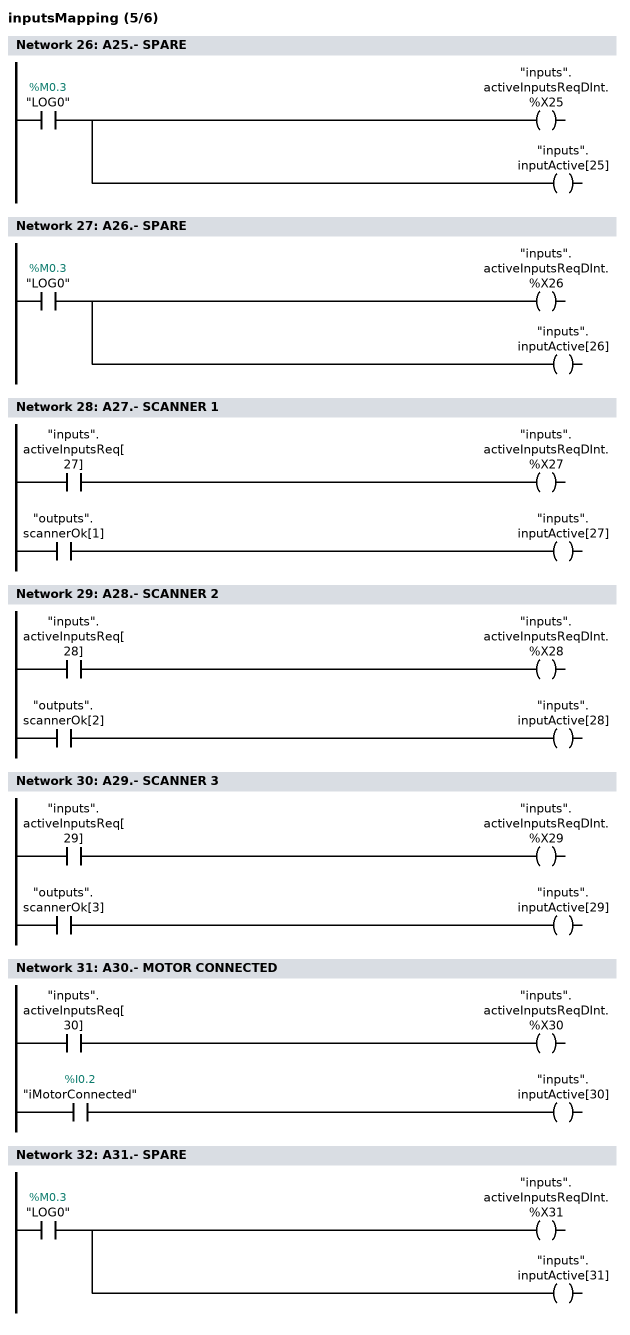
   RUNG wire#powerrail
      Contact( "LOG0" )
      wire#w1
      Coil( "inputs".activeInputsReqDInt.%X25 )
   END_RUNG
   RUNG wire#w1
      Coil( "inputs".inputActive[25] )
   END_RUNG
   // the same network as SCL:
   "inputs".activeInputsReqDInt.%X25 := "LOG0";
   "inputs".inputActive[25] := "LOG0";
END_REGION

REGION Network 27: A26.- SPARE
   RUNG wire#powerrail
      Contact( "LOG0" )
      wire#w1
      Coil( "inputs".activeInputsReqDInt.%X26 )
   END_RUNG
   RUNG wire#w1
      Coil( "inputs".inputActive[26] )
   END_RUNG
   // the same network as SCL:
   "inputs".activeInputsReqDInt.%X26 := "LOG0";
   "inputs".inputActive[26] := "LOG0";
END_REGION

REGION Network 28: A27.- SCANNER 1
   RUNG wire#powerrail
      Contact( "inputs".activeInputsReq[27] )
      Coil( "inputs".activeInputsReqDInt.%X27 )
   END_RUNG
   RUNG wire#powerrail
      Contact( "outputs".scannerOk[1] )
      Coil( "inputs".inputActive[27] )
   END_RUNG
   // the same network as SCL:
   "inputs".activeInputsReqDInt.%X27 := "inputs".activeInputsReq[27];
   "inputs".inputActive[27] := "outputs".scannerOk[1];
END_REGION

REGION Network 29: A28.- SCANNER 2
   RUNG wire#powerrail
      Contact( "inputs".activeInputsReq[28] )
      Coil( "inputs".activeInputsReqDInt.%X28 )
   END_RUNG
   RUNG wire#powerrail
      Contact( "outputs".scannerOk[2] )
      Coil( "inputs".inputActive[28] )
   END_RUNG
   // the same network as SCL:
   "inputs".activeInputsReqDInt.%X28 := "inputs".activeInputsReq[28];
   "inputs".inputActive[28] := "outputs".scannerOk[2];
END_REGION

REGION Network 30: A29.- SCANNER 3
   RUNG wire#powerrail
      Contact( "inputs".activeInputsReq[29] )
      Coil( "inputs".activeInputsReqDInt.%X29 )
   END_RUNG
   RUNG wire#powerrail
      Contact( "outputs".scannerOk[3] )
      Coil( "inputs".inputActive[29] )
   END_RUNG
   // the same network as SCL:
   "inputs".activeInputsReqDInt.%X29 := "inputs".activeInputsReq[29];
   "inputs".inputActive[29] := "outputs".scannerOk[3];
END_REGION

REGION Network 31: A30.- MOTOR CONNECTED
   RUNG wire#powerrail
      Contact( "inputs".activeInputsReq[30] )
      Coil( "inputs".activeInputsReqDInt.%X30 )
   END_RUNG
   RUNG wire#powerrail
      Contact( "iMotorConnected" )
      Coil( "inputs".inputActive[30] )
   END_RUNG
   // the same network as SCL:
   "inputs".activeInputsReqDInt.%X30 := "inputs".activeInputsReq[30];
   "inputs".inputActive[30] := "iMotorConnected";
END_REGION

REGION Network 32: A31.- SPARE
   RUNG wire#powerrail
      Contact( "LOG0" )
      wire#w1
      Coil( "inputs".activeInputsReqDInt.%X31 )
   END_RUNG
   RUNG wire#w1
      Coil( "inputs".inputActive[31] )
   END_RUNG
   // the same network as SCL:
   "inputs".activeInputsReqDInt.%X31 := "LOG0";
   "inputs".inputActive[31] := "LOG0";
END_REGION

REGION Network 33: HMI SENSOR OVERVIEW
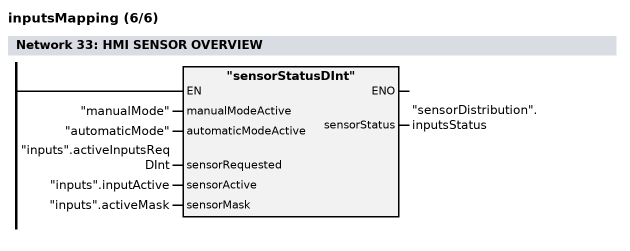
   RUNG wire#powerrail
      "sensorStatusDInt"(manualModeActive := "manualMode", automaticModeActive := "automaticMode", sensorRequested := "inputs".activeInputsReqDInt, sensorActive := "inputs".inputActive, sensorMask := "inputs".activeMask, sensorStatus => "sensorDistribution".inputsStatus)
   END_RUNG
   // the same network as SCL:
   "sensorStatusDInt"(manualModeActive := "manualMode",
                      automaticModeActive := "automaticMode",
                      sensorRequested := "inputs".activeInputsReqDInt,
                      sensorActive := "inputs".inputActive,
                      sensorMask := "inputs".activeMask,
                      sensorStatus => "sensorDistribution".inputsStatus);
END_REGION
END_FUNCTION

FUNCTION "sensorStatusDInt" : Void   // FC37, LAD
{ S7_Optimized_Access := 'TRUE' }
VERSION : 0.1
// stored: AutoNumber true, IsIECCheckEnabled false, SetENOAutomatically false, UDAEnableTagReadback false
   VAR_INPUT
      manualModeActive : Bool;
      automaticModeActive : Bool;
      sensorRequested : DInt;
      sensorActive : Array[0..31] of Bool;
      sensorMask : Array[0..31] of Bool;
   END_VAR
   VAR_OUTPUT
      sensorStatus : Array[0..31] of Byte;
   END_VAR
BEGIN

REGION Network 1: Status 0
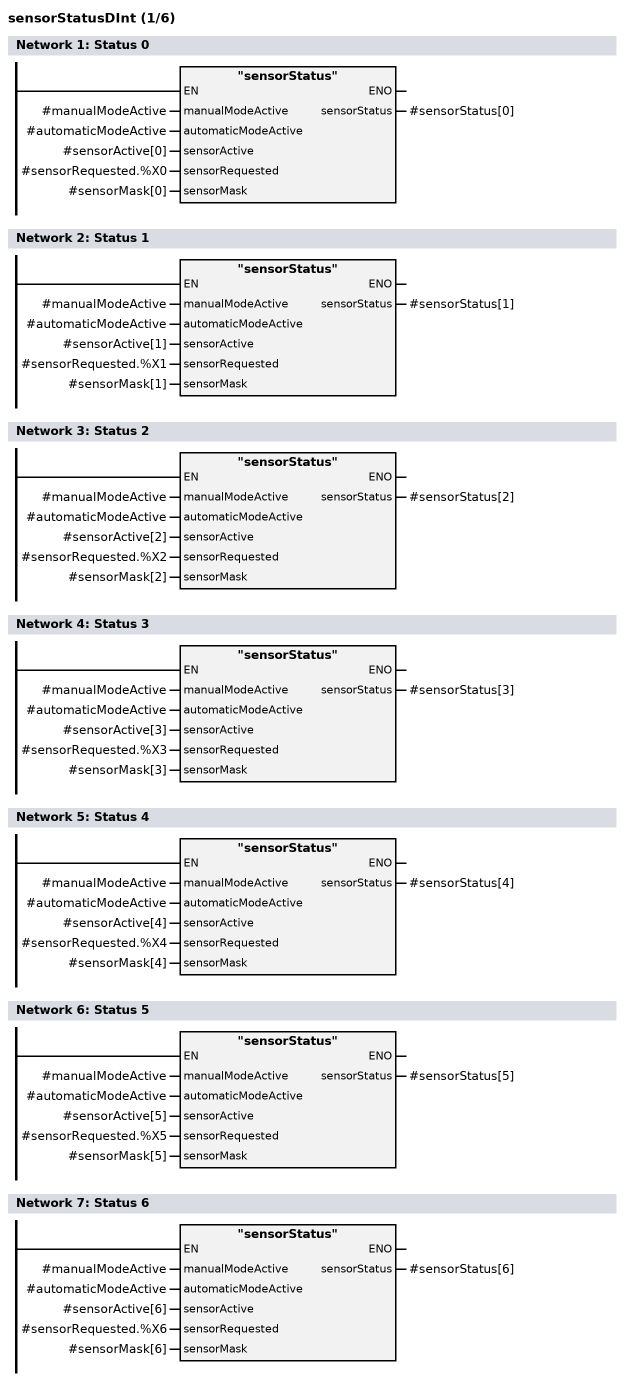
   RUNG wire#powerrail
      "sensorStatus"(manualModeActive := #manualModeActive, automaticModeActive := #automaticModeActive, sensorActive := #sensorActive[0], sensorRequested := #sensorRequested.%X0, sensorMask := #sensorMask[0], sensorStatus => #sensorStatus[0])
   END_RUNG
   // the same network as SCL:
   "sensorStatus"(manualModeActive := #manualModeActive,
                  automaticModeActive := #automaticModeActive,
                  sensorActive := #sensorActive[0],
                  sensorRequested := #sensorRequested.%X0,
                  sensorMask := #sensorMask[0],
                  sensorStatus => #sensorStatus[0]);
END_REGION

REGION Network 2: Status 1
   RUNG wire#powerrail
      "sensorStatus"(manualModeActive := #manualModeActive, automaticModeActive := #automaticModeActive, sensorActive := #sensorActive[1], sensorRequested := #sensorRequested.%X1, sensorMask := #sensorMask[1], sensorStatus => #sensorStatus[1])
   END_RUNG
   // the same network as SCL:
   "sensorStatus"(manualModeActive := #manualModeActive,
                  automaticModeActive := #automaticModeActive,
                  sensorActive := #sensorActive[1],
                  sensorRequested := #sensorRequested.%X1,
                  sensorMask := #sensorMask[1],
                  sensorStatus => #sensorStatus[1]);
END_REGION

REGION Network 3: Status 2
   RUNG wire#powerrail
      "sensorStatus"(manualModeActive := #manualModeActive, automaticModeActive := #automaticModeActive, sensorActive := #sensorActive[2], sensorRequested := #sensorRequested.%X2, sensorMask := #sensorMask[2], sensorStatus => #sensorStatus[2])
   END_RUNG
   // the same network as SCL:
   "sensorStatus"(manualModeActive := #manualModeActive,
                  automaticModeActive := #automaticModeActive,
                  sensorActive := #sensorActive[2],
                  sensorRequested := #sensorRequested.%X2,
                  sensorMask := #sensorMask[2],
                  sensorStatus => #sensorStatus[2]);
END_REGION

REGION Network 4: Status 3
   RUNG wire#powerrail
      "sensorStatus"(manualModeActive := #manualModeActive, automaticModeActive := #automaticModeActive, sensorActive := #sensorActive[3], sensorRequested := #sensorRequested.%X3, sensorMask := #sensorMask[3], sensorStatus => #sensorStatus[3])
   END_RUNG
   // the same network as SCL:
   "sensorStatus"(manualModeActive := #manualModeActive,
                  automaticModeActive := #automaticModeActive,
                  sensorActive := #sensorActive[3],
                  sensorRequested := #sensorRequested.%X3,
                  sensorMask := #sensorMask[3],
                  sensorStatus => #sensorStatus[3]);
END_REGION

REGION Network 5: Status 4
   RUNG wire#powerrail
      "sensorStatus"(manualModeActive := #manualModeActive, automaticModeActive := #automaticModeActive, sensorActive := #sensorActive[4], sensorRequested := #sensorRequested.%X4, sensorMask := #sensorMask[4], sensorStatus => #sensorStatus[4])
   END_RUNG
   // the same network as SCL:
   "sensorStatus"(manualModeActive := #manualModeActive,
                  automaticModeActive := #automaticModeActive,
                  sensorActive := #sensorActive[4],
                  sensorRequested := #sensorRequested.%X4,
                  sensorMask := #sensorMask[4],
                  sensorStatus => #sensorStatus[4]);
END_REGION

REGION Network 6: Status 5
   RUNG wire#powerrail
      "sensorStatus"(manualModeActive := #manualModeActive, automaticModeActive := #automaticModeActive, sensorActive := #sensorActive[5], sensorRequested := #sensorRequested.%X5, sensorMask := #sensorMask[5], sensorStatus => #sensorStatus[5])
   END_RUNG
   // the same network as SCL:
   "sensorStatus"(manualModeActive := #manualModeActive,
                  automaticModeActive := #automaticModeActive,
                  sensorActive := #sensorActive[5],
                  sensorRequested := #sensorRequested.%X5,
                  sensorMask := #sensorMask[5],
                  sensorStatus => #sensorStatus[5]);
END_REGION

REGION Network 7: Status 6
   RUNG wire#powerrail
      "sensorStatus"(manualModeActive := #manualModeActive, automaticModeActive := #automaticModeActive, sensorActive := #sensorActive[6], sensorRequested := #sensorRequested.%X6, sensorMask := #sensorMask[6], sensorStatus => #sensorStatus[6])
   END_RUNG
   // the same network as SCL:
   "sensorStatus"(manualModeActive := #manualModeActive,
                  automaticModeActive := #automaticModeActive,
                  sensorActive := #sensorActive[6],
                  sensorRequested := #sensorRequested.%X6,
                  sensorMask := #sensorMask[6],
                  sensorStatus => #sensorStatus[6]);
END_REGION

REGION Network 8: Status 7
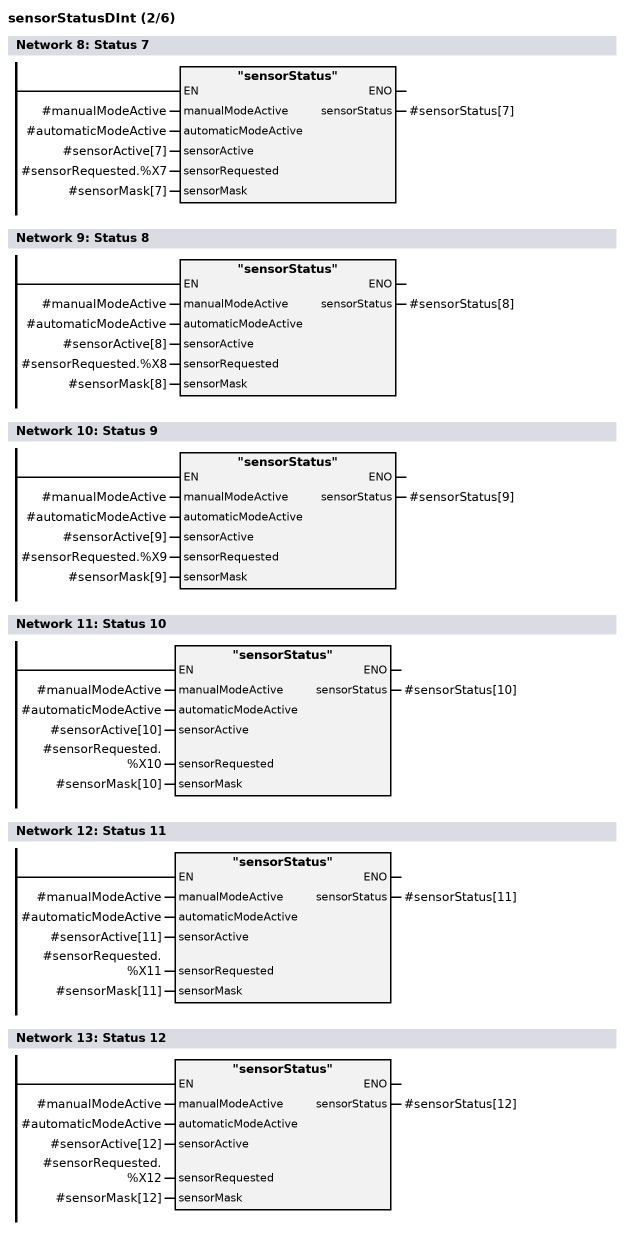
   RUNG wire#powerrail
      "sensorStatus"(manualModeActive := #manualModeActive, automaticModeActive := #automaticModeActive, sensorActive := #sensorActive[7], sensorRequested := #sensorRequested.%X7, sensorMask := #sensorMask[7], sensorStatus => #sensorStatus[7])
   END_RUNG
   // the same network as SCL:
   "sensorStatus"(manualModeActive := #manualModeActive,
                  automaticModeActive := #automaticModeActive,
                  sensorActive := #sensorActive[7],
                  sensorRequested := #sensorRequested.%X7,
                  sensorMask := #sensorMask[7],
                  sensorStatus => #sensorStatus[7]);
END_REGION

REGION Network 9: Status 8
   RUNG wire#powerrail
      "sensorStatus"(manualModeActive := #manualModeActive, automaticModeActive := #automaticModeActive, sensorActive := #sensorActive[8], sensorRequested := #sensorRequested.%X8, sensorMask := #sensorMask[8], sensorStatus => #sensorStatus[8])
   END_RUNG
   // the same network as SCL:
   "sensorStatus"(manualModeActive := #manualModeActive,
                  automaticModeActive := #automaticModeActive,
                  sensorActive := #sensorActive[8],
                  sensorRequested := #sensorRequested.%X8,
                  sensorMask := #sensorMask[8],
                  sensorStatus => #sensorStatus[8]);
END_REGION

REGION Network 10: Status 9
   RUNG wire#powerrail
      "sensorStatus"(manualModeActive := #manualModeActive, automaticModeActive := #automaticModeActive, sensorActive := #sensorActive[9], sensorRequested := #sensorRequested.%X9, sensorMask := #sensorMask[9], sensorStatus => #sensorStatus[9])
   END_RUNG
   // the same network as SCL:
   "sensorStatus"(manualModeActive := #manualModeActive,
                  automaticModeActive := #automaticModeActive,
                  sensorActive := #sensorActive[9],
                  sensorRequested := #sensorRequested.%X9,
                  sensorMask := #sensorMask[9],
                  sensorStatus => #sensorStatus[9]);
END_REGION

REGION Network 11: Status 10
   RUNG wire#powerrail
      "sensorStatus"(manualModeActive := #manualModeActive, automaticModeActive := #automaticModeActive, sensorActive := #sensorActive[10], sensorRequested := #sensorRequested.%X10, sensorMask := #sensorMask[10], sensorStatus => #sensorStatus[10])
   END_RUNG
   // the same network as SCL:
   "sensorStatus"(manualModeActive := #manualModeActive,
                  automaticModeActive := #automaticModeActive,
                  sensorActive := #sensorActive[10],
                  sensorRequested := #sensorRequested.%X10,
                  sensorMask := #sensorMask[10],
                  sensorStatus => #sensorStatus[10]);
END_REGION

REGION Network 12: Status 11
   RUNG wire#powerrail
      "sensorStatus"(manualModeActive := #manualModeActive, automaticModeActive := #automaticModeActive, sensorActive := #sensorActive[11], sensorRequested := #sensorRequested.%X11, sensorMask := #sensorMask[11], sensorStatus => #sensorStatus[11])
   END_RUNG
   // the same network as SCL:
   "sensorStatus"(manualModeActive := #manualModeActive,
                  automaticModeActive := #automaticModeActive,
                  sensorActive := #sensorActive[11],
                  sensorRequested := #sensorRequested.%X11,
                  sensorMask := #sensorMask[11],
                  sensorStatus => #sensorStatus[11]);
END_REGION

REGION Network 13: Status 12
   RUNG wire#powerrail
      "sensorStatus"(manualModeActive := #manualModeActive, automaticModeActive := #automaticModeActive, sensorActive := #sensorActive[12], sensorRequested := #sensorRequested.%X12, sensorMask := #sensorMask[12], sensorStatus => #sensorStatus[12])
   END_RUNG
   // the same network as SCL:
   "sensorStatus"(manualModeActive := #manualModeActive,
                  automaticModeActive := #automaticModeActive,
                  sensorActive := #sensorActive[12],
                  sensorRequested := #sensorRequested.%X12,
                  sensorMask := #sensorMask[12],
                  sensorStatus => #sensorStatus[12]);
END_REGION

REGION Network 14: Status 13
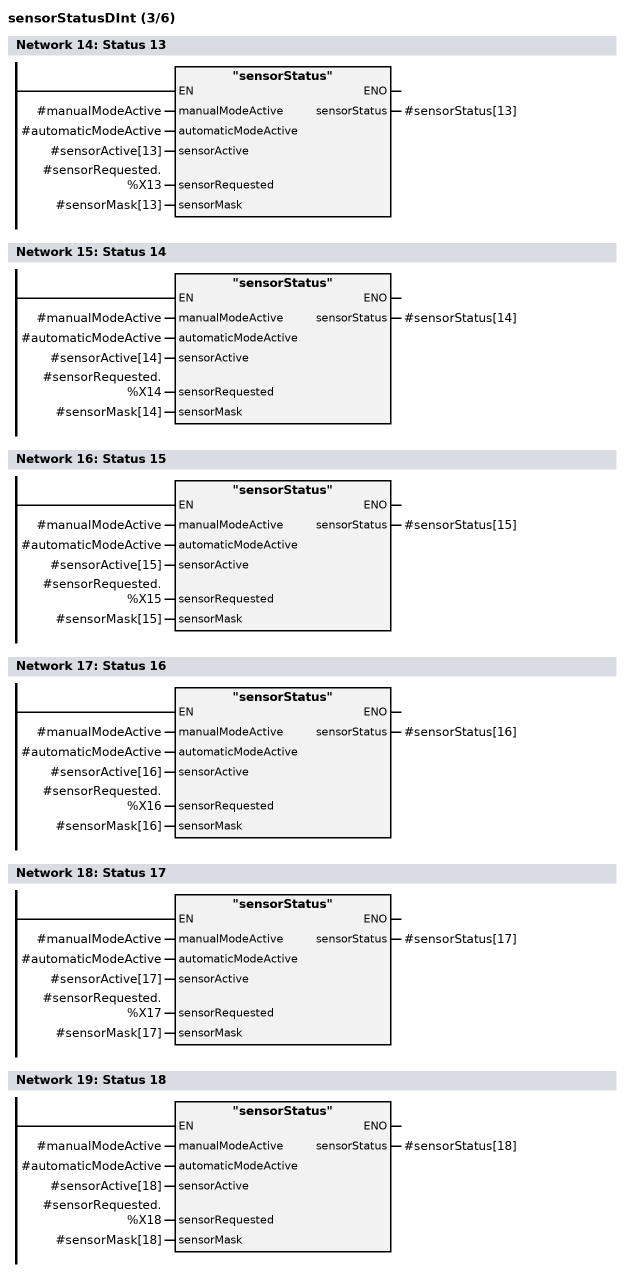
   RUNG wire#powerrail
      "sensorStatus"(manualModeActive := #manualModeActive, automaticModeActive := #automaticModeActive, sensorActive := #sensorActive[13], sensorRequested := #sensorRequested.%X13, sensorMask := #sensorMask[13], sensorStatus => #sensorStatus[13])
   END_RUNG
   // the same network as SCL:
   "sensorStatus"(manualModeActive := #manualModeActive,
                  automaticModeActive := #automaticModeActive,
                  sensorActive := #sensorActive[13],
                  sensorRequested := #sensorRequested.%X13,
                  sensorMask := #sensorMask[13],
                  sensorStatus => #sensorStatus[13]);
END_REGION

REGION Network 15: Status 14
   RUNG wire#powerrail
      "sensorStatus"(manualModeActive := #manualModeActive, automaticModeActive := #automaticModeActive, sensorActive := #sensorActive[14], sensorRequested := #sensorRequested.%X14, sensorMask := #sensorMask[14], sensorStatus => #sensorStatus[14])
   END_RUNG
   // the same network as SCL:
   "sensorStatus"(manualModeActive := #manualModeActive,
                  automaticModeActive := #automaticModeActive,
                  sensorActive := #sensorActive[14],
                  sensorRequested := #sensorRequested.%X14,
                  sensorMask := #sensorMask[14],
                  sensorStatus => #sensorStatus[14]);
END_REGION

REGION Network 16: Status 15
   RUNG wire#powerrail
      "sensorStatus"(manualModeActive := #manualModeActive, automaticModeActive := #automaticModeActive, sensorActive := #sensorActive[15], sensorRequested := #sensorRequested.%X15, sensorMask := #sensorMask[15], sensorStatus => #sensorStatus[15])
   END_RUNG
   // the same network as SCL:
   "sensorStatus"(manualModeActive := #manualModeActive,
                  automaticModeActive := #automaticModeActive,
                  sensorActive := #sensorActive[15],
                  sensorRequested := #sensorRequested.%X15,
                  sensorMask := #sensorMask[15],
                  sensorStatus => #sensorStatus[15]);
END_REGION

REGION Network 17: Status 16
   RUNG wire#powerrail
      "sensorStatus"(manualModeActive := #manualModeActive, automaticModeActive := #automaticModeActive, sensorActive := #sensorActive[16], sensorRequested := #sensorRequested.%X16, sensorMask := #sensorMask[16], sensorStatus => #sensorStatus[16])
   END_RUNG
   // the same network as SCL:
   "sensorStatus"(manualModeActive := #manualModeActive,
                  automaticModeActive := #automaticModeActive,
                  sensorActive := #sensorActive[16],
                  sensorRequested := #sensorRequested.%X16,
                  sensorMask := #sensorMask[16],
                  sensorStatus => #sensorStatus[16]);
END_REGION

REGION Network 18: Status 17
   RUNG wire#powerrail
      "sensorStatus"(manualModeActive := #manualModeActive, automaticModeActive := #automaticModeActive, sensorActive := #sensorActive[17], sensorRequested := #sensorRequested.%X17, sensorMask := #sensorMask[17], sensorStatus => #sensorStatus[17])
   END_RUNG
   // the same network as SCL:
   "sensorStatus"(manualModeActive := #manualModeActive,
                  automaticModeActive := #automaticModeActive,
                  sensorActive := #sensorActive[17],
                  sensorRequested := #sensorRequested.%X17,
                  sensorMask := #sensorMask[17],
                  sensorStatus => #sensorStatus[17]);
END_REGION

REGION Network 19: Status 18
   RUNG wire#powerrail
      "sensorStatus"(manualModeActive := #manualModeActive, automaticModeActive := #automaticModeActive, sensorActive := #sensorActive[18], sensorRequested := #sensorRequested.%X18, sensorMask := #sensorMask[18], sensorStatus => #sensorStatus[18])
   END_RUNG
   // the same network as SCL:
   "sensorStatus"(manualModeActive := #manualModeActive,
                  automaticModeActive := #automaticModeActive,
                  sensorActive := #sensorActive[18],
                  sensorRequested := #sensorRequested.%X18,
                  sensorMask := #sensorMask[18],
                  sensorStatus => #sensorStatus[18]);
END_REGION

REGION Network 20: Status 19
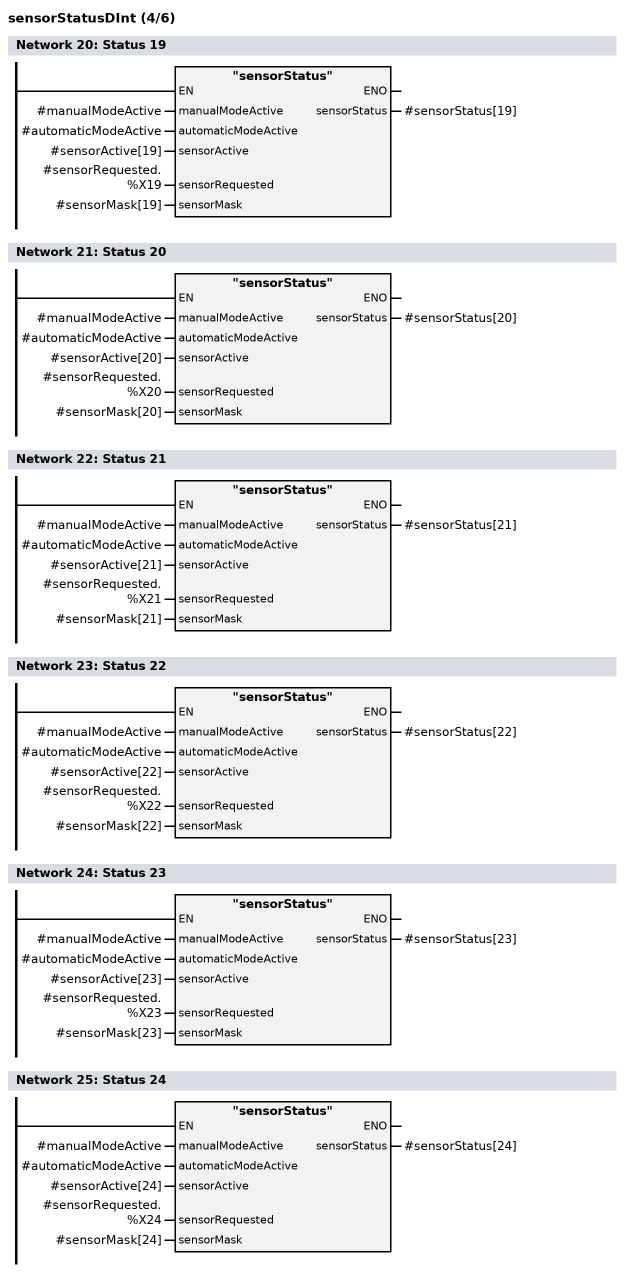
   RUNG wire#powerrail
      "sensorStatus"(manualModeActive := #manualModeActive, automaticModeActive := #automaticModeActive, sensorActive := #sensorActive[19], sensorRequested := #sensorRequested.%X19, sensorMask := #sensorMask[19], sensorStatus => #sensorStatus[19])
   END_RUNG
   // the same network as SCL:
   "sensorStatus"(manualModeActive := #manualModeActive,
                  automaticModeActive := #automaticModeActive,
                  sensorActive := #sensorActive[19],
                  sensorRequested := #sensorRequested.%X19,
                  sensorMask := #sensorMask[19],
                  sensorStatus => #sensorStatus[19]);
END_REGION

REGION Network 21: Status 20
   RUNG wire#powerrail
      "sensorStatus"(manualModeActive := #manualModeActive, automaticModeActive := #automaticModeActive, sensorActive := #sensorActive[20], sensorRequested := #sensorRequested.%X20, sensorMask := #sensorMask[20], sensorStatus => #sensorStatus[20])
   END_RUNG
   // the same network as SCL:
   "sensorStatus"(manualModeActive := #manualModeActive,
                  automaticModeActive := #automaticModeActive,
                  sensorActive := #sensorActive[20],
                  sensorRequested := #sensorRequested.%X20,
                  sensorMask := #sensorMask[20],
                  sensorStatus => #sensorStatus[20]);
END_REGION

REGION Network 22: Status 21
   RUNG wire#powerrail
      "sensorStatus"(manualModeActive := #manualModeActive, automaticModeActive := #automaticModeActive, sensorActive := #sensorActive[21], sensorRequested := #sensorRequested.%X21, sensorMask := #sensorMask[21], sensorStatus => #sensorStatus[21])
   END_RUNG
   // the same network as SCL:
   "sensorStatus"(manualModeActive := #manualModeActive,
                  automaticModeActive := #automaticModeActive,
                  sensorActive := #sensorActive[21],
                  sensorRequested := #sensorRequested.%X21,
                  sensorMask := #sensorMask[21],
                  sensorStatus => #sensorStatus[21]);
END_REGION

REGION Network 23: Status 22
   RUNG wire#powerrail
      "sensorStatus"(manualModeActive := #manualModeActive, automaticModeActive := #automaticModeActive, sensorActive := #sensorActive[22], sensorRequested := #sensorRequested.%X22, sensorMask := #sensorMask[22], sensorStatus => #sensorStatus[22])
   END_RUNG
   // the same network as SCL:
   "sensorStatus"(manualModeActive := #manualModeActive,
                  automaticModeActive := #automaticModeActive,
                  sensorActive := #sensorActive[22],
                  sensorRequested := #sensorRequested.%X22,
                  sensorMask := #sensorMask[22],
                  sensorStatus => #sensorStatus[22]);
END_REGION

REGION Network 24: Status 23
   RUNG wire#powerrail
      "sensorStatus"(manualModeActive := #manualModeActive, automaticModeActive := #automaticModeActive, sensorActive := #sensorActive[23], sensorRequested := #sensorRequested.%X23, sensorMask := #sensorMask[23], sensorStatus => #sensorStatus[23])
   END_RUNG
   // the same network as SCL:
   "sensorStatus"(manualModeActive := #manualModeActive,
                  automaticModeActive := #automaticModeActive,
                  sensorActive := #sensorActive[23],
                  sensorRequested := #sensorRequested.%X23,
                  sensorMask := #sensorMask[23],
                  sensorStatus => #sensorStatus[23]);
END_REGION

REGION Network 25: Status 24
   RUNG wire#powerrail
      "sensorStatus"(manualModeActive := #manualModeActive, automaticModeActive := #automaticModeActive, sensorActive := #sensorActive[24], sensorRequested := #sensorRequested.%X24, sensorMask := #sensorMask[24], sensorStatus => #sensorStatus[24])
   END_RUNG
   // the same network as SCL:
   "sensorStatus"(manualModeActive := #manualModeActive,
                  automaticModeActive := #automaticModeActive,
                  sensorActive := #sensorActive[24],
                  sensorRequested := #sensorRequested.%X24,
                  sensorMask := #sensorMask[24],
                  sensorStatus => #sensorStatus[24]);
END_REGION

REGION Network 26: Status 25
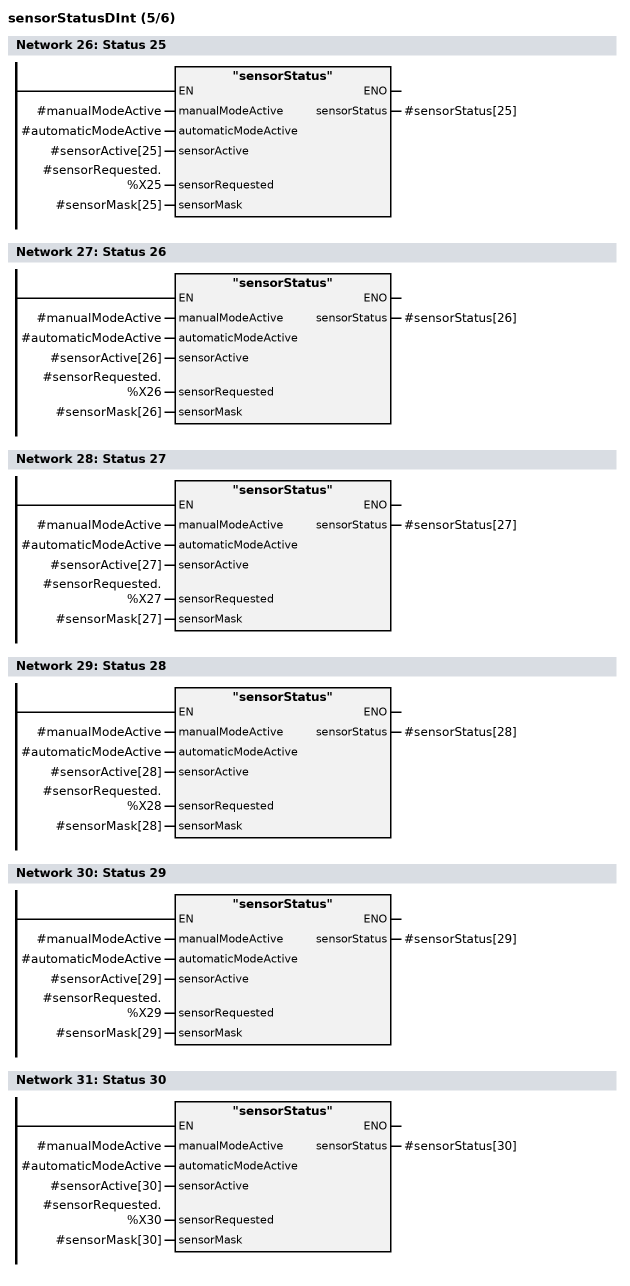
   RUNG wire#powerrail
      "sensorStatus"(manualModeActive := #manualModeActive, automaticModeActive := #automaticModeActive, sensorActive := #sensorActive[25], sensorRequested := #sensorRequested.%X25, sensorMask := #sensorMask[25], sensorStatus => #sensorStatus[25])
   END_RUNG
   // the same network as SCL:
   "sensorStatus"(manualModeActive := #manualModeActive,
                  automaticModeActive := #automaticModeActive,
                  sensorActive := #sensorActive[25],
                  sensorRequested := #sensorRequested.%X25,
                  sensorMask := #sensorMask[25],
                  sensorStatus => #sensorStatus[25]);
END_REGION

REGION Network 27: Status 26
   RUNG wire#powerrail
      "sensorStatus"(manualModeActive := #manualModeActive, automaticModeActive := #automaticModeActive, sensorActive := #sensorActive[26], sensorRequested := #sensorRequested.%X26, sensorMask := #sensorMask[26], sensorStatus => #sensorStatus[26])
   END_RUNG
   // the same network as SCL:
   "sensorStatus"(manualModeActive := #manualModeActive,
                  automaticModeActive := #automaticModeActive,
                  sensorActive := #sensorActive[26],
                  sensorRequested := #sensorRequested.%X26,
                  sensorMask := #sensorMask[26],
                  sensorStatus => #sensorStatus[26]);
END_REGION

REGION Network 28: Status 27
   RUNG wire#powerrail
      "sensorStatus"(manualModeActive := #manualModeActive, automaticModeActive := #automaticModeActive, sensorActive := #sensorActive[27], sensorRequested := #sensorRequested.%X27, sensorMask := #sensorMask[27], sensorStatus => #sensorStatus[27])
   END_RUNG
   // the same network as SCL:
   "sensorStatus"(manualModeActive := #manualModeActive,
                  automaticModeActive := #automaticModeActive,
                  sensorActive := #sensorActive[27],
                  sensorRequested := #sensorRequested.%X27,
                  sensorMask := #sensorMask[27],
                  sensorStatus => #sensorStatus[27]);
END_REGION

REGION Network 29: Status 28
   RUNG wire#powerrail
      "sensorStatus"(manualModeActive := #manualModeActive, automaticModeActive := #automaticModeActive, sensorActive := #sensorActive[28], sensorRequested := #sensorRequested.%X28, sensorMask := #sensorMask[28], sensorStatus => #sensorStatus[28])
   END_RUNG
   // the same network as SCL:
   "sensorStatus"(manualModeActive := #manualModeActive,
                  automaticModeActive := #automaticModeActive,
                  sensorActive := #sensorActive[28],
                  sensorRequested := #sensorRequested.%X28,
                  sensorMask := #sensorMask[28],
                  sensorStatus => #sensorStatus[28]);
END_REGION

REGION Network 30: Status 29
   RUNG wire#powerrail
      "sensorStatus"(manualModeActive := #manualModeActive, automaticModeActive := #automaticModeActive, sensorActive := #sensorActive[29], sensorRequested := #sensorRequested.%X29, sensorMask := #sensorMask[29], sensorStatus => #sensorStatus[29])
   END_RUNG
   // the same network as SCL:
   "sensorStatus"(manualModeActive := #manualModeActive,
                  automaticModeActive := #automaticModeActive,
                  sensorActive := #sensorActive[29],
                  sensorRequested := #sensorRequested.%X29,
                  sensorMask := #sensorMask[29],
                  sensorStatus => #sensorStatus[29]);
END_REGION

REGION Network 31: Status 30
   RUNG wire#powerrail
      "sensorStatus"(manualModeActive := #manualModeActive, automaticModeActive := #automaticModeActive, sensorActive := #sensorActive[30], sensorRequested := #sensorRequested.%X30, sensorMask := #sensorMask[30], sensorStatus => #sensorStatus[30])
   END_RUNG
   // the same network as SCL:
   "sensorStatus"(manualModeActive := #manualModeActive,
                  automaticModeActive := #automaticModeActive,
                  sensorActive := #sensorActive[30],
                  sensorRequested := #sensorRequested.%X30,
                  sensorMask := #sensorMask[30],
                  sensorStatus => #sensorStatus[30]);
END_REGION

REGION Network 32: Status 31
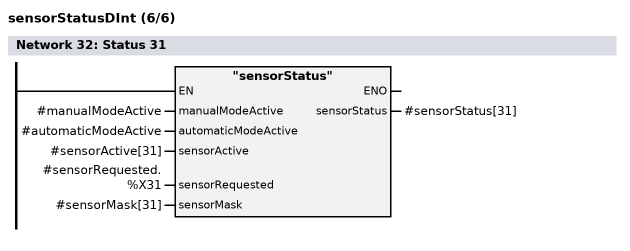
   RUNG wire#powerrail
      "sensorStatus"(manualModeActive := #manualModeActive, automaticModeActive := #automaticModeActive, sensorActive := #sensorActive[31], sensorRequested := #sensorRequested.%X31, sensorMask := #sensorMask[31], sensorStatus => #sensorStatus[31])
   END_RUNG
   // the same network as SCL:
   "sensorStatus"(manualModeActive := #manualModeActive,
                  automaticModeActive := #automaticModeActive,
                  sensorActive := #sensorActive[31],
                  sensorRequested := #sensorRequested.%X31,
                  sensorMask := #sensorMask[31],
                  sensorStatus => #sensorStatus[31]);
END_REGION
END_FUNCTION

FUNCTION "sensorStatus" : Void   // FC36, LAD
{ S7_Optimized_Access := 'TRUE' }
VERSION : 0.1
// stored: AutoNumber true, IsIECCheckEnabled false, SetENOAutomatically false, UDAEnableTagReadback false
   VAR_INPUT
      manualModeActive : Bool;
      automaticModeActive : Bool;
      sensorActive : Bool;
      sensorRequested : Bool;
      sensorMask : Bool;
   END_VAR
   VAR_OUTPUT
      sensorStatus : Int;
   END_VAR
   VAR_TEMP
      localMask : Bool;
   END_VAR
BEGIN

REGION Network 1
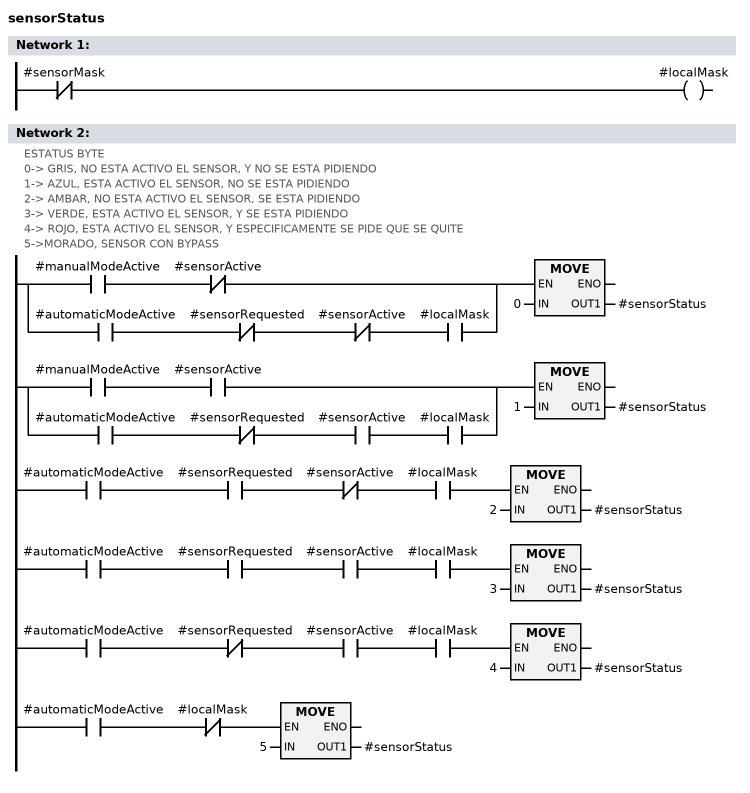
   RUNG wire#powerrail
      I_Contact( #sensorMask )
      Coil( #localMask )
   END_RUNG
   // the same network as SCL:
   #localMask := NOT #sensorMask;
END_REGION

REGION Network 2
   // ESTATUS BYTE
   // 0-> GRIS, NO ESTA ACTIVO EL SENSOR, Y NO SE ESTA PIDIENDO
   // 1-> AZUL, ESTA ACTIVO EL SENSOR, NO SE ESTA PIDIENDO
   // 2-> AMBAR, NO ESTA ACTIVO EL SENSOR, SE ESTA PIDIENDO
   // 3-> VERDE, ESTA ACTIVO EL SENSOR, Y SE ESTA PIDIENDO
   // 4-> ROJO, ESTA ACTIVO EL SENSOR, Y ESPECIFICAMENTE SE PIDE QUE SE QUITE
   // 5->MORADO, SENSOR CON BYPASS
   RUNG wire#powerrail
      Contact( #manualModeActive )
      I_Contact( #sensorActive )
      wire#w1
      Move(in := 0, out1 => #sensorStatus)
   END_RUNG
   RUNG wire#powerrail
      Contact( #automaticModeActive )
      I_Contact( #sensorRequested )
      I_Contact( #sensorActive )
      Contact( #localMask )
   END_RUNG wire#w1
   RUNG wire#powerrail
      Contact( #manualModeActive )
      Contact( #sensorActive )
      wire#w2
      Move(in := 1, out1 => #sensorStatus)
   END_RUNG
   RUNG wire#powerrail
      Contact( #automaticModeActive )
      I_Contact( #sensorRequested )
      Contact( #sensorActive )
      Contact( #localMask )
   END_RUNG wire#w2
   RUNG wire#powerrail
      Contact( #automaticModeActive )
      Contact( #sensorRequested )
      I_Contact( #sensorActive )
      Contact( #localMask )
      Move(in := 2, out1 => #sensorStatus)
   END_RUNG
   RUNG wire#powerrail
      Contact( #automaticModeActive )
      Contact( #sensorRequested )
      Contact( #sensorActive )
      Contact( #localMask )
      Move(in := 3, out1 => #sensorStatus)
   END_RUNG
   RUNG wire#powerrail
      Contact( #automaticModeActive )
      I_Contact( #sensorRequested )
      Contact( #sensorActive )
      Contact( #localMask )
      Move(in := 4, out1 => #sensorStatus)
   END_RUNG
   RUNG wire#powerrail
      Contact( #automaticModeActive )
      I_Contact( #localMask )
      Move(in := 5, out1 => #sensorStatus)
   END_RUNG
   // the same network as SCL:
   IF (#manualModeActive AND NOT #sensorActive) OR (#automaticModeActive AND NOT #sensorRequested AND NOT #sensorActive AND #localMask) THEN
       #sensorStatus := 0;
   END_IF;
   IF (#manualModeActive AND #sensorActive) OR (#automaticModeActive AND NOT #sensorRequested AND #sensorActive AND #localMask) THEN
       #sensorStatus := 1;
   END_IF;
   IF #automaticModeActive AND #sensorRequested AND NOT #sensorActive AND #localMask THEN
       #sensorStatus := 2;
   END_IF;
   IF #automaticModeActive AND #sensorRequested AND #sensorActive AND #localMask THEN
       #sensorStatus := 3;
   END_IF;
   IF #automaticModeActive AND NOT #sensorRequested AND #sensorActive AND #localMask THEN
       #sensorStatus := 4;
   END_IF;
   IF #automaticModeActive AND NOT #localMask THEN #sensorStatus := 5; END_IF;
END_REGION
END_FUNCTION

FUNCTION "cylinderControl" : Void   // FC9, LAD
{ S7_Optimized_Access := 'TRUE' }
VERSION : 0.1
// stored: AutoNumber true, IsIECCheckEnabled false, SetENOAutomatically false, UDAEnableTagReadback false
   VAR_TEMP
      leftTrackReady : Bool;
      rightTrackReady : Bool;
      plasticBridgeReady : Bool;
      retractLocatingPinReady : Bool;
      enableCylinders : Bool;
      retractClampsReady : Bool;
   END_VAR
   VAR_TEMP   // added for the SCL form of the ladder/FBD networks
      _w1 : Bool;
   END_VAR
BEGIN

REGION Network 1: ENABLE CYLINDER GLOBAL
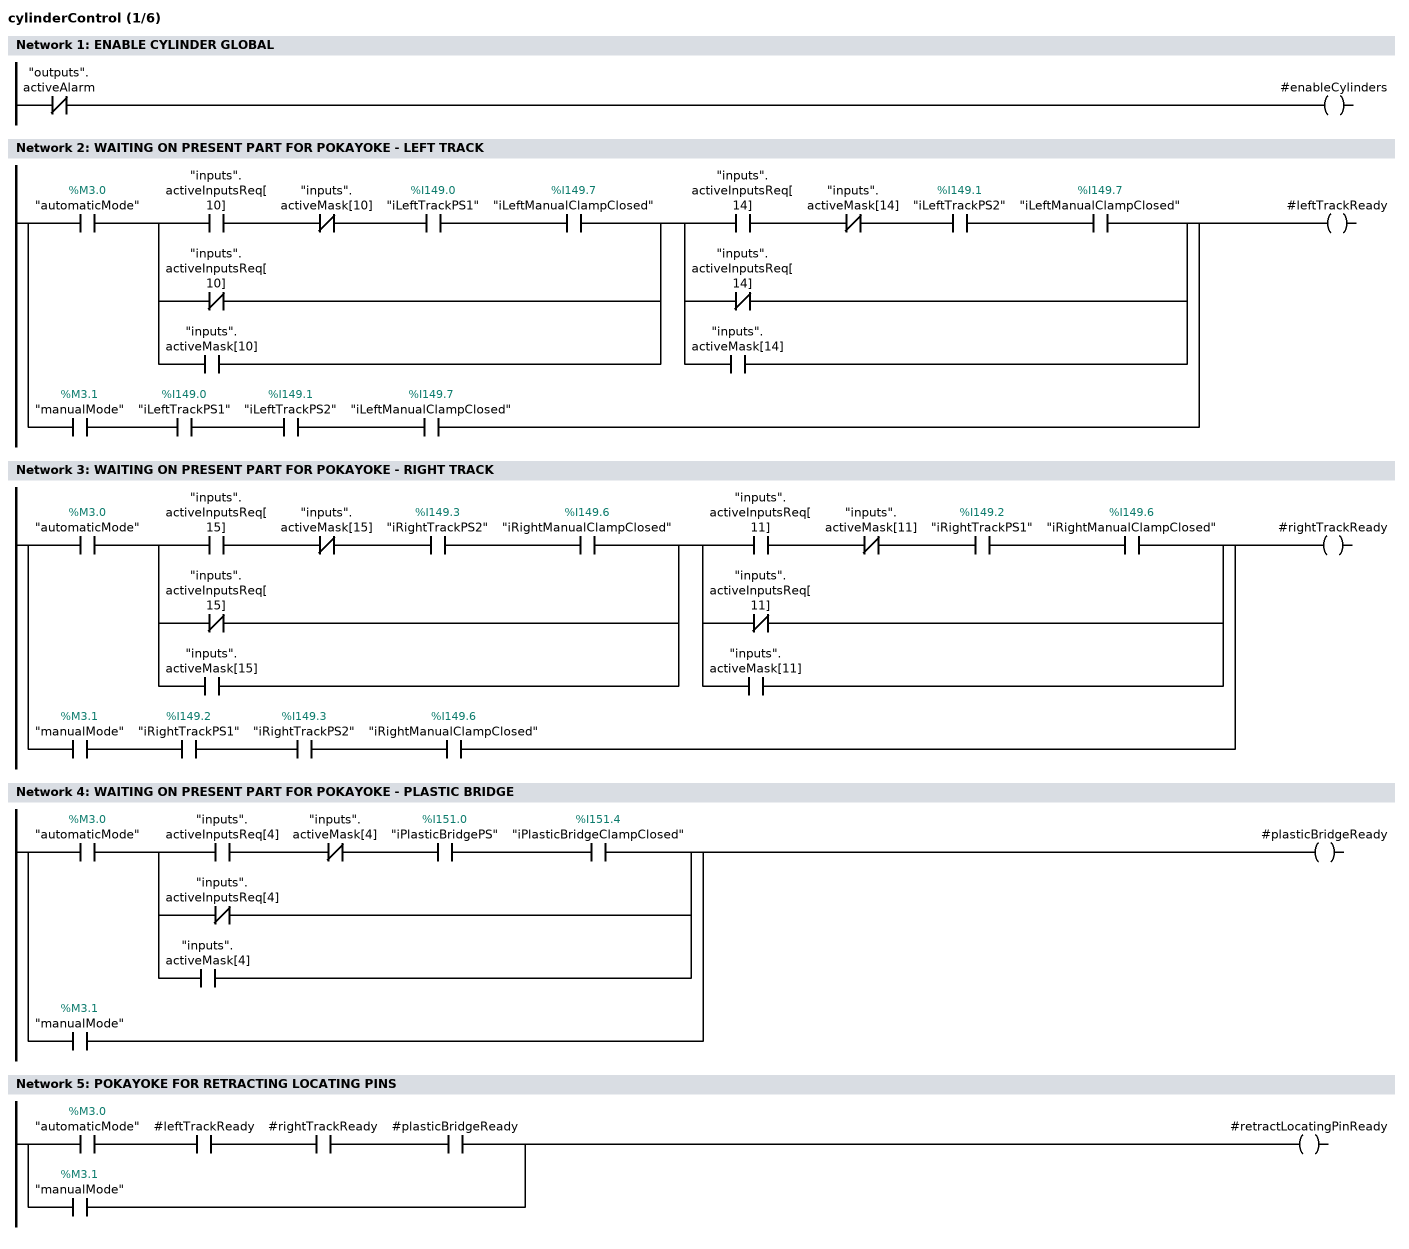
   RUNG wire#powerrail
      I_Contact( "outputs".activeAlarm )
      Coil( #enableCylinders )
   END_RUNG
   // the same network as SCL:
   #enableCylinders := NOT "outputs".activeAlarm;
END_REGION

REGION Network 2: WAITING ON PRESENT PART FOR POKAYOKE - LEFT TRACK
   RUNG wire#powerrail
      Contact( "automaticMode" )
      wire#w1
      Contact( "inputs".activeInputsReq[10] )
      I_Contact( "inputs".activeMask[10] )
      Contact( "iLeftTrackPS1" )
      Contact( "iLeftManualClampClosed" )
      wire#w2
      Contact( "inputs".activeInputsReq[14] )
      I_Contact( "inputs".activeMask[14] )
      Contact( "iLeftTrackPS2" )
      Contact( "iLeftManualClampClosed" )
      wire#w3
      Coil( #leftTrackReady )
   END_RUNG
   RUNG wire#w1
      I_Contact( "inputs".activeInputsReq[10] )
   END_RUNG wire#w2
   RUNG wire#w1
      Contact( "inputs".activeMask[10] )
   END_RUNG wire#w2
   RUNG wire#w2
      I_Contact( "inputs".activeInputsReq[14] )
   END_RUNG wire#w3
   RUNG wire#w2
      Contact( "inputs".activeMask[14] )
   END_RUNG wire#w3
   RUNG wire#powerrail
      Contact( "manualMode" )
      Contact( "iLeftTrackPS1" )
      Contact( "iLeftTrackPS2" )
      Contact( "iLeftManualClampClosed" )
   END_RUNG wire#w3
   // the same network as SCL:
   #leftTrackReady := ("automaticMode" AND (("inputs".activeInputsReq[10] AND NOT "inputs".activeMask[10] AND "iLeftTrackPS1" AND "iLeftManualClampClosed") OR NOT "inputs".activeInputsReq[10] OR "inputs".activeMask[10]) AND (("inputs".activeInputsReq[14] AND NOT "inputs".activeMask[14] AND "iLeftTrackPS2" AND "iLeftManualClampClosed") OR NOT "inputs".activeInputsReq[14] OR "inputs".activeMask[14])) OR ("manualMode" AND "iLeftTrackPS1" AND "iLeftTrackPS2" AND "iLeftManualClampClosed");
END_REGION

REGION Network 3: WAITING ON PRESENT PART FOR POKAYOKE - RIGHT TRACK
   RUNG wire#powerrail
      Contact( "automaticMode" )
      wire#w1
      Contact( "inputs".activeInputsReq[15] )
      I_Contact( "inputs".activeMask[15] )
      Contact( "iRightTrackPS2" )
      Contact( "iRightManualClampClosed" )
      wire#w2
      Contact( "inputs".activeInputsReq[11] )
      I_Contact( "inputs".activeMask[11] )
      Contact( "iRightTrackPS1" )
      Contact( "iRightManualClampClosed" )
      wire#w3
      Coil( #rightTrackReady )
   END_RUNG
   RUNG wire#w1
      I_Contact( "inputs".activeInputsReq[15] )
   END_RUNG wire#w2
   RUNG wire#w1
      Contact( "inputs".activeMask[15] )
   END_RUNG wire#w2
   RUNG wire#w2
      I_Contact( "inputs".activeInputsReq[11] )
   END_RUNG wire#w3
   RUNG wire#w2
      Contact( "inputs".activeMask[11] )
   END_RUNG wire#w3
   RUNG wire#powerrail
      Contact( "manualMode" )
      Contact( "iRightTrackPS1" )
      Contact( "iRightTrackPS2" )
      Contact( "iRightManualClampClosed" )
   END_RUNG wire#w3
   // the same network as SCL:
   #rightTrackReady := ("automaticMode" AND (("inputs".activeInputsReq[15] AND NOT "inputs".activeMask[15] AND "iRightTrackPS2" AND "iRightManualClampClosed") OR NOT "inputs".activeInputsReq[15] OR "inputs".activeMask[15]) AND (("inputs".activeInputsReq[11] AND NOT "inputs".activeMask[11] AND "iRightTrackPS1" AND "iRightManualClampClosed") OR NOT "inputs".activeInputsReq[11] OR "inputs".activeMask[11])) OR ("manualMode" AND "iRightTrackPS1" AND "iRightTrackPS2" AND "iRightManualClampClosed");
END_REGION

REGION Network 4: WAITING ON PRESENT PART FOR POKAYOKE - PLASTIC BRIDGE
   RUNG wire#powerrail
      Contact( "automaticMode" )
      wire#w1
      Contact( "inputs".activeInputsReq[4] )
      I_Contact( "inputs".activeMask[4] )
      Contact( "iPlasticBridgePS" )
      Contact( "iPlasticBridgeClampClosed" )
      wire#w2
      Coil( #plasticBridgeReady )
   END_RUNG
   RUNG wire#w1
      I_Contact( "inputs".activeInputsReq[4] )
   END_RUNG wire#w2
   RUNG wire#w1
      Contact( "inputs".activeMask[4] )
   END_RUNG wire#w2
   RUNG wire#powerrail
      Contact( "manualMode" )
   END_RUNG wire#w2
   // the same network as SCL:
   #plasticBridgeReady := ("automaticMode" AND (("inputs".activeInputsReq[4] AND NOT "inputs".activeMask[4] AND "iPlasticBridgePS" AND "iPlasticBridgeClampClosed") OR NOT "inputs".activeInputsReq[4] OR "inputs".activeMask[4])) OR "manualMode";
END_REGION

REGION Network 5: POKAYOKE FOR RETRACTING LOCATING PINS
   RUNG wire#powerrail
      Contact( "automaticMode" )
      Contact( #leftTrackReady )
      Contact( #rightTrackReady )
      Contact( #plasticBridgeReady )
      wire#w1
      Coil( #retractLocatingPinReady )
   END_RUNG
   RUNG wire#powerrail
      Contact( "manualMode" )
   END_RUNG wire#w1
   // the same network as SCL:
   #retractLocatingPinReady := ("automaticMode" AND #leftTrackReady AND #rightTrackReady AND #plasticBridgeReady) OR "manualMode";
END_REGION

REGION Network 6: POKAYOKE FOR RETRACTING CLAMPS
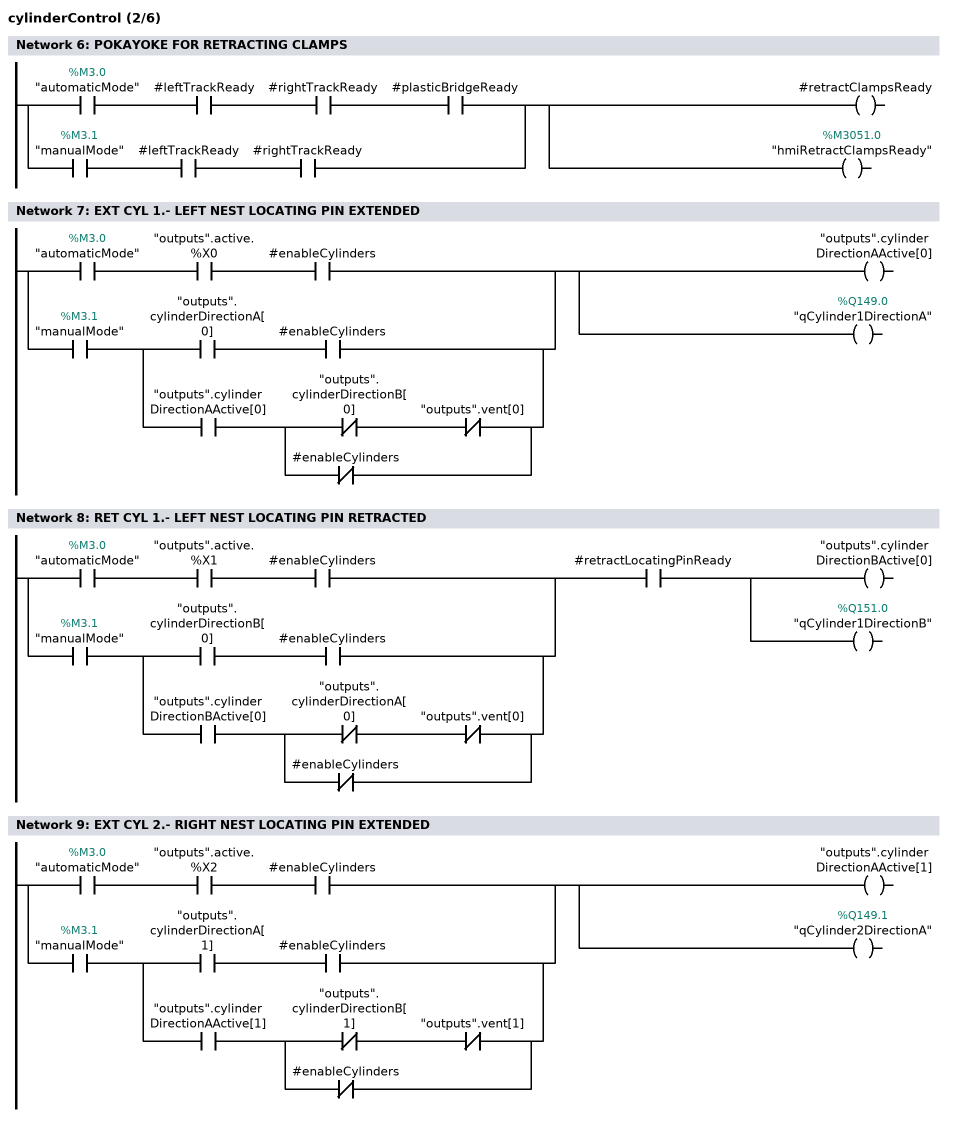
   RUNG wire#powerrail
      Contact( "automaticMode" )
      Contact( #leftTrackReady )
      Contact( #rightTrackReady )
      Contact( #plasticBridgeReady )
      wire#w1
      Coil( #retractClampsReady )
   END_RUNG
   RUNG wire#powerrail
      Contact( "manualMode" )
      Contact( #leftTrackReady )
      Contact( #rightTrackReady )
   END_RUNG wire#w1
   RUNG wire#w1
      Coil( "hmiRetractClampsReady" )
   END_RUNG
   // the same network as SCL:
   #retractClampsReady := ("automaticMode" AND #leftTrackReady AND #rightTrackReady AND #plasticBridgeReady) OR ("manualMode" AND #leftTrackReady AND #rightTrackReady);
   "hmiRetractClampsReady" := #retractClampsReady;
END_REGION

REGION Network 7: EXT CYL 1.- LEFT NEST LOCATING PIN EXTENDED
   RUNG wire#powerrail
      Contact( "automaticMode" )
      Contact( "outputs".active.%X0 )
      Contact( #enableCylinders )
      wire#w1
      Coil( "outputs".cylinderDirectionAActive[0] )
   END_RUNG
   RUNG wire#powerrail
      Contact( "manualMode" )
      wire#w2
      Contact( "outputs".cylinderDirectionA[0] )
      Contact( #enableCylinders )
   END_RUNG wire#w1
   RUNG wire#w2
      Contact( "outputs".cylinderDirectionAActive[0] )
      wire#w3
      I_Contact( "outputs".cylinderDirectionB[0] )
      I_Contact( "outputs".vent[0] )
   END_RUNG wire#w1
   RUNG wire#w3
      I_Contact( #enableCylinders )
   END_RUNG wire#w1
   RUNG wire#w1
      Coil( "qCylinder1DirectionA" )
   END_RUNG
   // the same network as SCL:
   #_w1 := ("automaticMode" AND "outputs".active.%X0 AND #enableCylinders) OR ("manualMode" AND (("outputs".cylinderDirectionA[0] AND #enableCylinders) OR ("outputs".cylinderDirectionAActive[0] AND ((NOT "outputs".cylinderDirectionB[0] AND NOT "outputs".vent[0]) OR NOT #enableCylinders))));
   "outputs".cylinderDirectionAActive[0] := ("automaticMode" AND "outputs".active.%X0 AND #enableCylinders) OR ("manualMode" AND (("outputs".cylinderDirectionA[0] AND #enableCylinders) OR ("outputs".cylinderDirectionAActive[0] AND ((NOT "outputs".cylinderDirectionB[0] AND NOT "outputs".vent[0]) OR NOT #enableCylinders))));
   "qCylinder1DirectionA" := #_w1;
END_REGION

REGION Network 8: RET CYL 1.- LEFT NEST LOCATING PIN RETRACTED
   RUNG wire#powerrail
      Contact( "automaticMode" )
      Contact( "outputs".active.%X1 )
      Contact( #enableCylinders )
      wire#w1
      Contact( #retractLocatingPinReady )
      wire#w4
      Coil( "outputs".cylinderDirectionBActive[0] )
   END_RUNG
   RUNG wire#powerrail
      Contact( "manualMode" )
      wire#w2
      Contact( "outputs".cylinderDirectionB[0] )
      Contact( #enableCylinders )
   END_RUNG wire#w1
   RUNG wire#w2
      Contact( "outputs".cylinderDirectionBActive[0] )
      wire#w3
      I_Contact( "outputs".cylinderDirectionA[0] )
      I_Contact( "outputs".vent[0] )
   END_RUNG wire#w1
   RUNG wire#w3
      I_Contact( #enableCylinders )
   END_RUNG wire#w1
   RUNG wire#w4
      Coil( "qCylinder1DirectionB" )
   END_RUNG
   // the same network as SCL:
   #_w1 := (("automaticMode" AND "outputs".active.%X1 AND #enableCylinders) OR ("manualMode" AND (("outputs".cylinderDirectionB[0] AND #enableCylinders) OR ("outputs".cylinderDirectionBActive[0] AND ((NOT "outputs".cylinderDirectionA[0] AND NOT "outputs".vent[0]) OR NOT #enableCylinders))))) AND #retractLocatingPinReady;
   "outputs".cylinderDirectionBActive[0] := (("automaticMode" AND "outputs".active.%X1 AND #enableCylinders) OR ("manualMode" AND (("outputs".cylinderDirectionB[0] AND #enableCylinders) OR ("outputs".cylinderDirectionBActive[0] AND ((NOT "outputs".cylinderDirectionA[0] AND NOT "outputs".vent[0]) OR NOT #enableCylinders))))) AND #retractLocatingPinReady;
   "qCylinder1DirectionB" := #_w1;
END_REGION

REGION Network 9: EXT CYL 2.- RIGHT NEST LOCATING PIN EXTENDED
   RUNG wire#powerrail
      Contact( "automaticMode" )
      Contact( "outputs".active.%X2 )
      Contact( #enableCylinders )
      wire#w1
      Coil( "outputs".cylinderDirectionAActive[1] )
   END_RUNG
   RUNG wire#powerrail
      Contact( "manualMode" )
      wire#w2
      Contact( "outputs".cylinderDirectionA[1] )
      Contact( #enableCylinders )
   END_RUNG wire#w1
   RUNG wire#w2
      Contact( "outputs".cylinderDirectionAActive[1] )
      wire#w3
      I_Contact( "outputs".cylinderDirectionB[1] )
      I_Contact( "outputs".vent[1] )
   END_RUNG wire#w1
   RUNG wire#w3
      I_Contact( #enableCylinders )
   END_RUNG wire#w1
   RUNG wire#w1
      Coil( "qCylinder2DirectionA" )
   END_RUNG
   // the same network as SCL:
   #_w1 := ("automaticMode" AND "outputs".active.%X2 AND #enableCylinders) OR ("manualMode" AND (("outputs".cylinderDirectionA[1] AND #enableCylinders) OR ("outputs".cylinderDirectionAActive[1] AND ((NOT "outputs".cylinderDirectionB[1] AND NOT "outputs".vent[1]) OR NOT #enableCylinders))));
   "outputs".cylinderDirectionAActive[1] := ("automaticMode" AND "outputs".active.%X2 AND #enableCylinders) OR ("manualMode" AND (("outputs".cylinderDirectionA[1] AND #enableCylinders) OR ("outputs".cylinderDirectionAActive[1] AND ((NOT "outputs".cylinderDirectionB[1] AND NOT "outputs".vent[1]) OR NOT #enableCylinders))));
   "qCylinder2DirectionA" := #_w1;
END_REGION

REGION Network 10: RET CYL 2.- RIGHT NEST LOCATING PIN RETRACTED
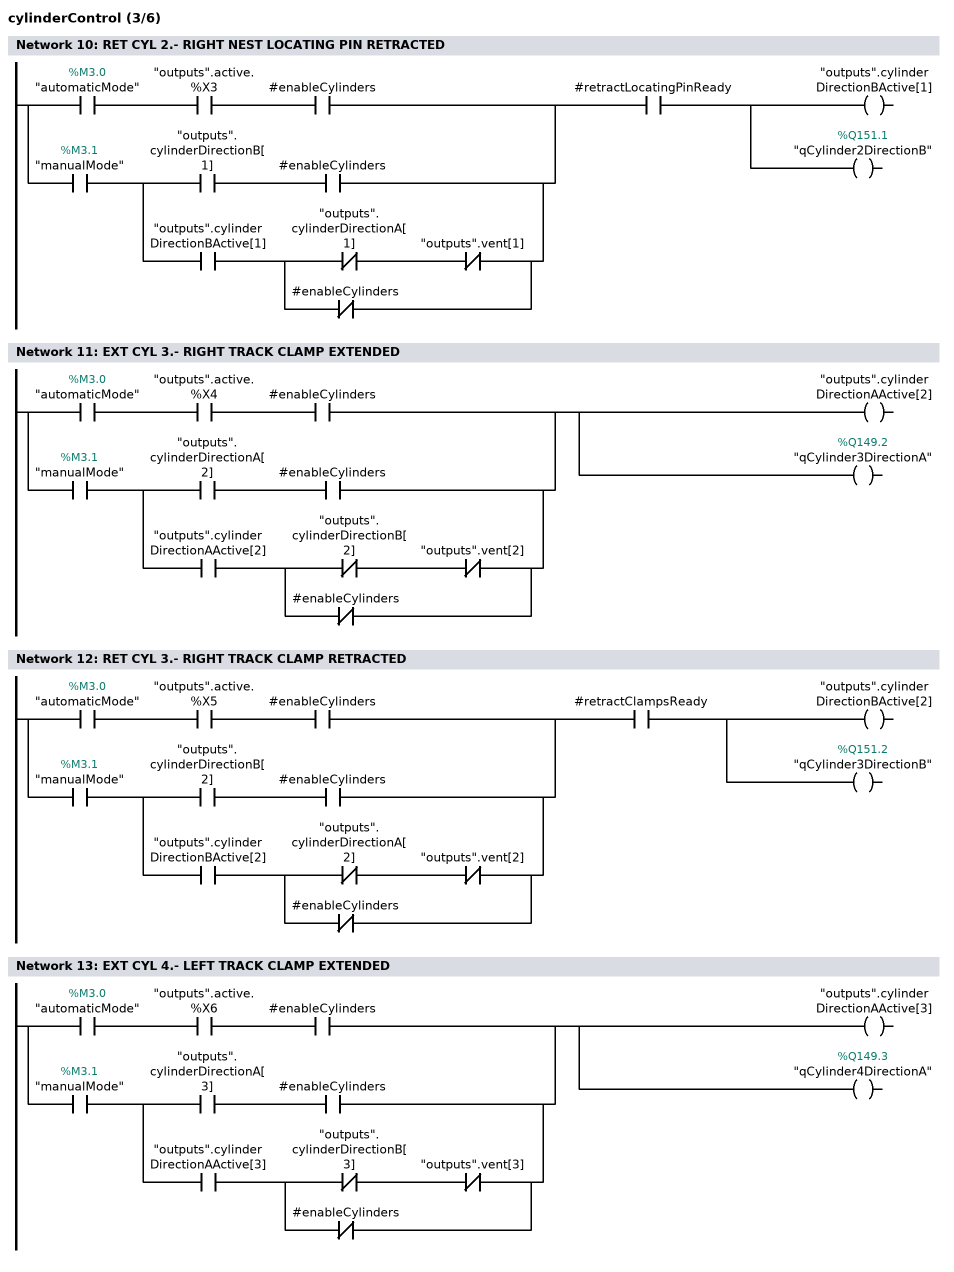
   RUNG wire#powerrail
      Contact( "automaticMode" )
      Contact( "outputs".active.%X3 )
      Contact( #enableCylinders )
      wire#w1
      Contact( #retractLocatingPinReady )
      wire#w4
      Coil( "outputs".cylinderDirectionBActive[1] )
   END_RUNG
   RUNG wire#powerrail
      Contact( "manualMode" )
      wire#w2
      Contact( "outputs".cylinderDirectionB[1] )
      Contact( #enableCylinders )
   END_RUNG wire#w1
   RUNG wire#w2
      Contact( "outputs".cylinderDirectionBActive[1] )
      wire#w3
      I_Contact( "outputs".cylinderDirectionA[1] )
      I_Contact( "outputs".vent[1] )
   END_RUNG wire#w1
   RUNG wire#w3
      I_Contact( #enableCylinders )
   END_RUNG wire#w1
   RUNG wire#w4
      Coil( "qCylinder2DirectionB" )
   END_RUNG
   // the same network as SCL:
   #_w1 := (("automaticMode" AND "outputs".active.%X3 AND #enableCylinders) OR ("manualMode" AND (("outputs".cylinderDirectionB[1] AND #enableCylinders) OR ("outputs".cylinderDirectionBActive[1] AND ((NOT "outputs".cylinderDirectionA[1] AND NOT "outputs".vent[1]) OR NOT #enableCylinders))))) AND #retractLocatingPinReady;
   "outputs".cylinderDirectionBActive[1] := (("automaticMode" AND "outputs".active.%X3 AND #enableCylinders) OR ("manualMode" AND (("outputs".cylinderDirectionB[1] AND #enableCylinders) OR ("outputs".cylinderDirectionBActive[1] AND ((NOT "outputs".cylinderDirectionA[1] AND NOT "outputs".vent[1]) OR NOT #enableCylinders))))) AND #retractLocatingPinReady;
   "qCylinder2DirectionB" := #_w1;
END_REGION

REGION Network 11: EXT CYL 3.- RIGHT TRACK CLAMP EXTENDED
   RUNG wire#powerrail
      Contact( "automaticMode" )
      Contact( "outputs".active.%X4 )
      Contact( #enableCylinders )
      wire#w1
      Coil( "outputs".cylinderDirectionAActive[2] )
   END_RUNG
   RUNG wire#powerrail
      Contact( "manualMode" )
      wire#w2
      Contact( "outputs".cylinderDirectionA[2] )
      Contact( #enableCylinders )
   END_RUNG wire#w1
   RUNG wire#w2
      Contact( "outputs".cylinderDirectionAActive[2] )
      wire#w3
      I_Contact( "outputs".cylinderDirectionB[2] )
      I_Contact( "outputs".vent[2] )
   END_RUNG wire#w1
   RUNG wire#w3
      I_Contact( #enableCylinders )
   END_RUNG wire#w1
   RUNG wire#w1
      Coil( "qCylinder3DirectionA" )
   END_RUNG
   // the same network as SCL:
   #_w1 := ("automaticMode" AND "outputs".active.%X4 AND #enableCylinders) OR ("manualMode" AND (("outputs".cylinderDirectionA[2] AND #enableCylinders) OR ("outputs".cylinderDirectionAActive[2] AND ((NOT "outputs".cylinderDirectionB[2] AND NOT "outputs".vent[2]) OR NOT #enableCylinders))));
   "outputs".cylinderDirectionAActive[2] := ("automaticMode" AND "outputs".active.%X4 AND #enableCylinders) OR ("manualMode" AND (("outputs".cylinderDirectionA[2] AND #enableCylinders) OR ("outputs".cylinderDirectionAActive[2] AND ((NOT "outputs".cylinderDirectionB[2] AND NOT "outputs".vent[2]) OR NOT #enableCylinders))));
   "qCylinder3DirectionA" := #_w1;
END_REGION

REGION Network 12: RET CYL 3.- RIGHT TRACK CLAMP RETRACTED
   RUNG wire#powerrail
      Contact( "automaticMode" )
      Contact( "outputs".active.%X5 )
      Contact( #enableCylinders )
      wire#w1
      Contact( #retractClampsReady )
      wire#w4
      Coil( "outputs".cylinderDirectionBActive[2] )
   END_RUNG
   RUNG wire#powerrail
      Contact( "manualMode" )
      wire#w2
      Contact( "outputs".cylinderDirectionB[2] )
      Contact( #enableCylinders )
   END_RUNG wire#w1
   RUNG wire#w2
      Contact( "outputs".cylinderDirectionBActive[2] )
      wire#w3
      I_Contact( "outputs".cylinderDirectionA[2] )
      I_Contact( "outputs".vent[2] )
   END_RUNG wire#w1
   RUNG wire#w3
      I_Contact( #enableCylinders )
   END_RUNG wire#w1
   RUNG wire#w4
      Coil( "qCylinder3DirectionB" )
   END_RUNG
   // the same network as SCL:
   #_w1 := (("automaticMode" AND "outputs".active.%X5 AND #enableCylinders) OR ("manualMode" AND (("outputs".cylinderDirectionB[2] AND #enableCylinders) OR ("outputs".cylinderDirectionBActive[2] AND ((NOT "outputs".cylinderDirectionA[2] AND NOT "outputs".vent[2]) OR NOT #enableCylinders))))) AND #retractClampsReady;
   "outputs".cylinderDirectionBActive[2] := (("automaticMode" AND "outputs".active.%X5 AND #enableCylinders) OR ("manualMode" AND (("outputs".cylinderDirectionB[2] AND #enableCylinders) OR ("outputs".cylinderDirectionBActive[2] AND ((NOT "outputs".cylinderDirectionA[2] AND NOT "outputs".vent[2]) OR NOT #enableCylinders))))) AND #retractClampsReady;
   "qCylinder3DirectionB" := #_w1;
END_REGION

REGION Network 13: EXT CYL 4.- LEFT TRACK CLAMP EXTENDED
   RUNG wire#powerrail
      Contact( "automaticMode" )
      Contact( "outputs".active.%X6 )
      Contact( #enableCylinders )
      wire#w1
      Coil( "outputs".cylinderDirectionAActive[3] )
   END_RUNG
   RUNG wire#powerrail
      Contact( "manualMode" )
      wire#w2
      Contact( "outputs".cylinderDirectionA[3] )
      Contact( #enableCylinders )
   END_RUNG wire#w1
   RUNG wire#w2
      Contact( "outputs".cylinderDirectionAActive[3] )
      wire#w3
      I_Contact( "outputs".cylinderDirectionB[3] )
      I_Contact( "outputs".vent[3] )
   END_RUNG wire#w1
   RUNG wire#w3
      I_Contact( #enableCylinders )
   END_RUNG wire#w1
   RUNG wire#w1
      Coil( "qCylinder4DirectionA" )
   END_RUNG
   // the same network as SCL:
   #_w1 := ("automaticMode" AND "outputs".active.%X6 AND #enableCylinders) OR ("manualMode" AND (("outputs".cylinderDirectionA[3] AND #enableCylinders) OR ("outputs".cylinderDirectionAActive[3] AND ((NOT "outputs".cylinderDirectionB[3] AND NOT "outputs".vent[3]) OR NOT #enableCylinders))));
   "outputs".cylinderDirectionAActive[3] := ("automaticMode" AND "outputs".active.%X6 AND #enableCylinders) OR ("manualMode" AND (("outputs".cylinderDirectionA[3] AND #enableCylinders) OR ("outputs".cylinderDirectionAActive[3] AND ((NOT "outputs".cylinderDirectionB[3] AND NOT "outputs".vent[3]) OR NOT #enableCylinders))));
   "qCylinder4DirectionA" := #_w1;
END_REGION

REGION Network 14: RET CYL 4.- LEFT TRACK CLAMP RETRACTED
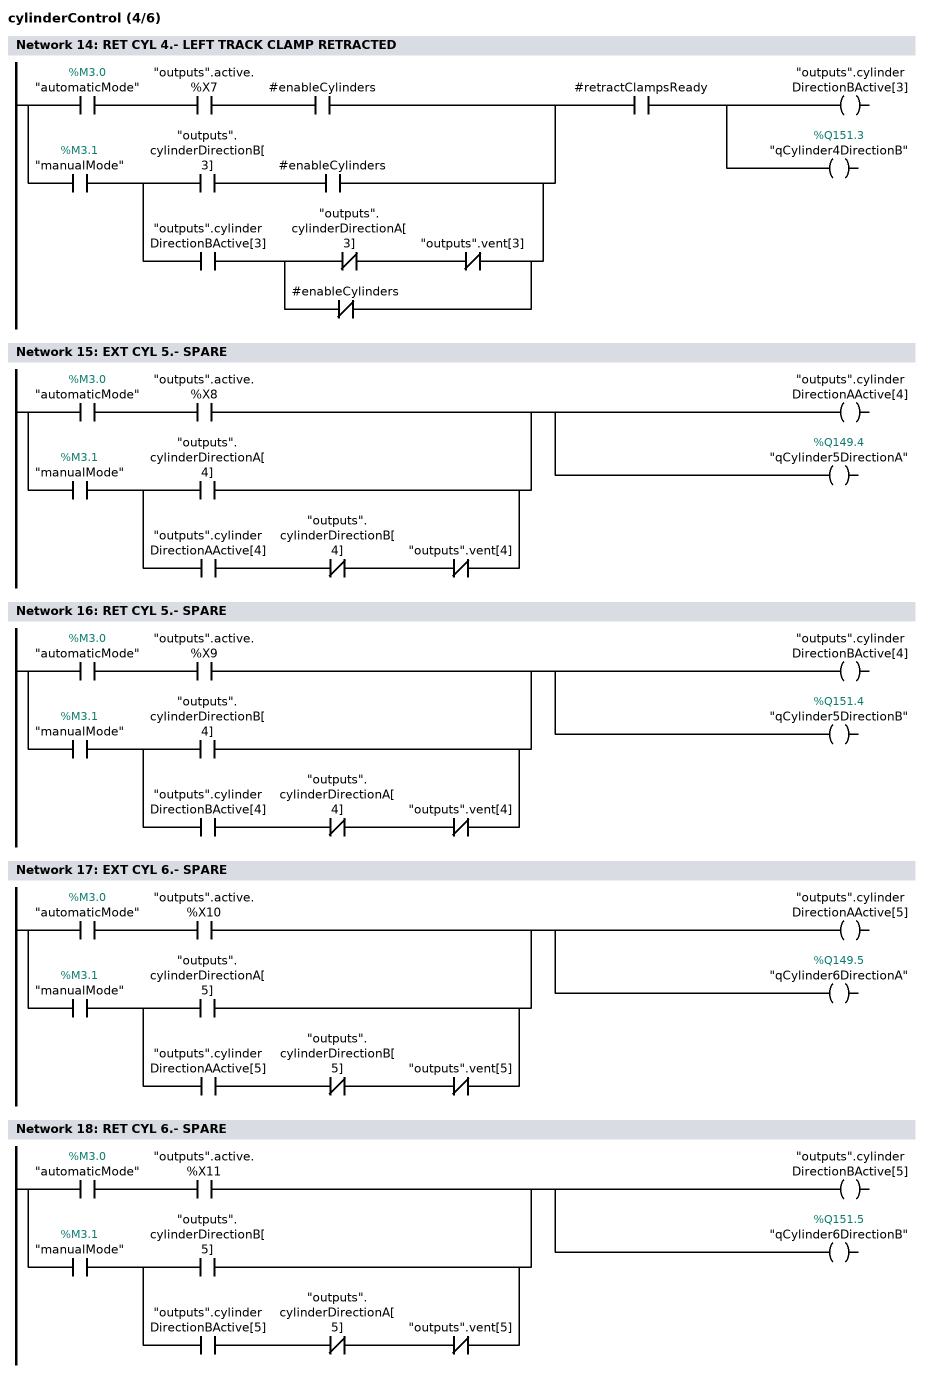
   RUNG wire#powerrail
      Contact( "automaticMode" )
      Contact( "outputs".active.%X7 )
      Contact( #enableCylinders )
      wire#w1
      Contact( #retractClampsReady )
      wire#w4
      Coil( "outputs".cylinderDirectionBActive[3] )
   END_RUNG
   RUNG wire#powerrail
      Contact( "manualMode" )
      wire#w2
      Contact( "outputs".cylinderDirectionB[3] )
      Contact( #enableCylinders )
   END_RUNG wire#w1
   RUNG wire#w2
      Contact( "outputs".cylinderDirectionBActive[3] )
      wire#w3
      I_Contact( "outputs".cylinderDirectionA[3] )
      I_Contact( "outputs".vent[3] )
   END_RUNG wire#w1
   RUNG wire#w3
      I_Contact( #enableCylinders )
   END_RUNG wire#w1
   RUNG wire#w4
      Coil( "qCylinder4DirectionB" )
   END_RUNG
   // the same network as SCL:
   #_w1 := (("automaticMode" AND "outputs".active.%X7 AND #enableCylinders) OR ("manualMode" AND (("outputs".cylinderDirectionB[3] AND #enableCylinders) OR ("outputs".cylinderDirectionBActive[3] AND ((NOT "outputs".cylinderDirectionA[3] AND NOT "outputs".vent[3]) OR NOT #enableCylinders))))) AND #retractClampsReady;
   "outputs".cylinderDirectionBActive[3] := (("automaticMode" AND "outputs".active.%X7 AND #enableCylinders) OR ("manualMode" AND (("outputs".cylinderDirectionB[3] AND #enableCylinders) OR ("outputs".cylinderDirectionBActive[3] AND ((NOT "outputs".cylinderDirectionA[3] AND NOT "outputs".vent[3]) OR NOT #enableCylinders))))) AND #retractClampsReady;
   "qCylinder4DirectionB" := #_w1;
END_REGION

REGION Network 15: EXT CYL 5.- SPARE
   RUNG wire#powerrail
      Contact( "automaticMode" )
      Contact( "outputs".active.%X8 )
      wire#w1
      Coil( "outputs".cylinderDirectionAActive[4] )
   END_RUNG
   RUNG wire#powerrail
      Contact( "manualMode" )
      wire#w2
      Contact( "outputs".cylinderDirectionA[4] )
   END_RUNG wire#w1
   RUNG wire#w2
      Contact( "outputs".cylinderDirectionAActive[4] )
      I_Contact( "outputs".cylinderDirectionB[4] )
      I_Contact( "outputs".vent[4] )
   END_RUNG wire#w1
   RUNG wire#w1
      Coil( "qCylinder5DirectionA" )
   END_RUNG
   // the same network as SCL:
   #_w1 := ("automaticMode" AND "outputs".active.%X8) OR ("manualMode" AND ("outputs".cylinderDirectionA[4] OR ("outputs".cylinderDirectionAActive[4] AND NOT "outputs".cylinderDirectionB[4] AND NOT "outputs".vent[4])));
   "outputs".cylinderDirectionAActive[4] := ("automaticMode" AND "outputs".active.%X8) OR ("manualMode" AND ("outputs".cylinderDirectionA[4] OR ("outputs".cylinderDirectionAActive[4] AND NOT "outputs".cylinderDirectionB[4] AND NOT "outputs".vent[4])));
   "qCylinder5DirectionA" := #_w1;
END_REGION

REGION Network 16: RET CYL 5.- SPARE
   RUNG wire#powerrail
      Contact( "automaticMode" )
      Contact( "outputs".active.%X9 )
      wire#w1
      Coil( "outputs".cylinderDirectionBActive[4] )
   END_RUNG
   RUNG wire#powerrail
      Contact( "manualMode" )
      wire#w2
      Contact( "outputs".cylinderDirectionB[4] )
   END_RUNG wire#w1
   RUNG wire#w2
      Contact( "outputs".cylinderDirectionBActive[4] )
      I_Contact( "outputs".cylinderDirectionA[4] )
      I_Contact( "outputs".vent[4] )
   END_RUNG wire#w1
   RUNG wire#w1
      Coil( "qCylinder5DirectionB" )
   END_RUNG
   // the same network as SCL:
   #_w1 := ("automaticMode" AND "outputs".active.%X9) OR ("manualMode" AND ("outputs".cylinderDirectionB[4] OR ("outputs".cylinderDirectionBActive[4] AND NOT "outputs".cylinderDirectionA[4] AND NOT "outputs".vent[4])));
   "outputs".cylinderDirectionBActive[4] := ("automaticMode" AND "outputs".active.%X9) OR ("manualMode" AND ("outputs".cylinderDirectionB[4] OR ("outputs".cylinderDirectionBActive[4] AND NOT "outputs".cylinderDirectionA[4] AND NOT "outputs".vent[4])));
   "qCylinder5DirectionB" := #_w1;
END_REGION

REGION Network 17: EXT CYL 6.- SPARE
   RUNG wire#powerrail
      Contact( "automaticMode" )
      Contact( "outputs".active.%X10 )
      wire#w1
      Coil( "outputs".cylinderDirectionAActive[5] )
   END_RUNG
   RUNG wire#powerrail
      Contact( "manualMode" )
      wire#w2
      Contact( "outputs".cylinderDirectionA[5] )
   END_RUNG wire#w1
   RUNG wire#w2
      Contact( "outputs".cylinderDirectionAActive[5] )
      I_Contact( "outputs".cylinderDirectionB[5] )
      I_Contact( "outputs".vent[5] )
   END_RUNG wire#w1
   RUNG wire#w1
      Coil( "qCylinder6DirectionA" )
   END_RUNG
   // the same network as SCL:
   #_w1 := ("automaticMode" AND "outputs".active.%X10) OR ("manualMode" AND ("outputs".cylinderDirectionA[5] OR ("outputs".cylinderDirectionAActive[5] AND NOT "outputs".cylinderDirectionB[5] AND NOT "outputs".vent[5])));
   "outputs".cylinderDirectionAActive[5] := ("automaticMode" AND "outputs".active.%X10) OR ("manualMode" AND ("outputs".cylinderDirectionA[5] OR ("outputs".cylinderDirectionAActive[5] AND NOT "outputs".cylinderDirectionB[5] AND NOT "outputs".vent[5])));
   "qCylinder6DirectionA" := #_w1;
END_REGION

REGION Network 18: RET CYL 6.- SPARE
   RUNG wire#powerrail
      Contact( "automaticMode" )
      Contact( "outputs".active.%X11 )
      wire#w1
      Coil( "outputs".cylinderDirectionBActive[5] )
   END_RUNG
   RUNG wire#powerrail
      Contact( "manualMode" )
      wire#w2
      Contact( "outputs".cylinderDirectionB[5] )
   END_RUNG wire#w1
   RUNG wire#w2
      Contact( "outputs".cylinderDirectionBActive[5] )
      I_Contact( "outputs".cylinderDirectionA[5] )
      I_Contact( "outputs".vent[5] )
   END_RUNG wire#w1
   RUNG wire#w1
      Coil( "qCylinder6DirectionB" )
   END_RUNG
   // the same network as SCL:
   #_w1 := ("automaticMode" AND "outputs".active.%X11) OR ("manualMode" AND ("outputs".cylinderDirectionB[5] OR ("outputs".cylinderDirectionBActive[5] AND NOT "outputs".cylinderDirectionA[5] AND NOT "outputs".vent[5])));
   "outputs".cylinderDirectionBActive[5] := ("automaticMode" AND "outputs".active.%X11) OR ("manualMode" AND ("outputs".cylinderDirectionB[5] OR ("outputs".cylinderDirectionBActive[5] AND NOT "outputs".cylinderDirectionA[5] AND NOT "outputs".vent[5])));
   "qCylinder6DirectionB" := #_w1;
END_REGION

REGION Network 19: EXT CYL 7.- SPARE
